LIN {X 0,Y 190.994,Z 614.523,A -85,B 0,C 180,E1 -21873.163,E2 -21873.163} C_VEL
LIN {X 0,Y 190.359,Z 618.573,A -85,B 0,C 180,E1 -21876.358,E2 -21876.358} C_VEL
LIN {X 0,Y 189.98,Z 620.669,A -85,B 0,C 180,E1 -21878.509,E2 -21878.509} C_VEL
LIN {X 0,Y 189.805,Z 622.334,A -85,B 0,C 180,E1 -21880.668,E2 -21880.668} C_VEL
LIN {X 0,Y 189.783,Z 623.59,A -85,B 0,C 180,E1 -21882.837,E2 -21882.837} C_VEL
LIN {X 0,Y 189.941,Z 624.591,A -85,B 0,C 180,E1 -21885.84,E2 -21885.84} C_VEL
LIN {X 0,Y 190.376,Z 624.78,A -85,B 0,C 180,E1 -21889.404,E2 -21889.404} C_VEL
LIN {X 0,Y 191.476,Z 623.671,A -85,B 0,C 180,E1 -21893.421,E2 -21893.421} C_VEL
LIN {X 0,Y 192.56,Z 622.169,A -85,B 0,C 180,E1 -21895.973,E2 -21895.973} C_VEL
LIN {X 0,Y 194.335,Z 619.447,A -85,B 0,C 180,E1 -21899.131,E2 -21899.131} C_VEL
LIN {X 0,Y 196.821,Z 615.459,A -85,B 0,C 180,E1 -21902.384,E2 -21902.384} C_VEL
LIN {X 0,Y 199.68,Z 610.497,A -85,B 0,C 180,E1 -21905.398,E2 -21905.398} C_VEL
LIN {X 0,Y 203.214,Z 603.837,A -85,B 0,C 180,E1 -21908.499,E2 -21908.499} C_VEL
LIN {X 0,Y 207.18,Z 595.882,A -85,B 0,C 180,E1 -21911.297,E2 -21911.297} C_VEL
LIN {X 0,Y 211.109,Z 587.168,A -85,B 0,C 180,E1 -21913.691,E2 -21913.691} C_VEL
LIN {X 0,Y 215.19,Z 576.766,A -85,B 0,C 180,E1 -21915.93,E2 -21915.93} C_VEL
LIN {X 0,Y 218.717,Z 566.352,A -85,B 0,C 180,E1 -21917.649,E2 -21917.649} C_VEL
LIN {X 0,Y 221.86,Z 554.889,A -85,B 0,C 180,E1 -21919.137,E2 -21919.137} C_VEL
LIN {X 0,Y 224.521,Z 543.286,A -85,B 0,C 180,E1 -21920.249,E2 -21920.249} C_VEL
LIN {X 0,Y 226.733,Z 530.168,A -85,B 0,C 180,E1 -21921.135,E2 -21921.135} C_VEL
LIN {X 0,Y 228.18,Z 516.758,A -85,B 0,C 180,E1 -21921.695,E2 -21921.695} C_VEL
LIN {X 0,Y 230.429,Z 476.831,A -85,B 0,C 180,E1 -21922.898,E2 -21922.898} C_VEL
LIN {X 0,Y 225.493,Z 465.84,A -85,B 0,C 180,E1 -21924.695,E2 -21924.695} C_VEL
LIN {X 0,Y 218.885,Z 453.171,A -85,B 0,C 180,E1 -21927.233,E2 -21927.233} C_VEL
LIN {X 0,Y 213.425,Z 444.071,A -85,B 0,C 180,E1 -21929.489,E2 -21929.489} C_VEL
LIN {X 0,Y 207.886,Z 435.651,A -85,B 0,C 180,E1 -21931.986,E2 -21931.986} C_VEL
LIN {X 0,Y 204.807,Z 431.149,A -85,B 0,C 180,E1 -21933.507,E2 -21933.507} C_VEL
LIN {X 0,Y 201.32,Z 426.295,A -85,B 0,C 180,E1 -21935.361,E2 -21935.361} C_VEL
LIN {X 0,Y 198.268,Z 423.081,A -85,B 0,C 180,E1 -21937.051,E2 -21937.051} C_VEL
LIN {X 0,Y 197.017,Z 420.675,A -85,B 0,C 180,E1 -21937.865,E2 -21937.865} C_VEL
LIN {X 0,Y 194.483,Z 418.918,A -85,B 0,C 180,E1 -21939.37,E2 -21939.37} C_VEL
LIN {X 0,Y 193.045,Z 416.552,A -85,B 0,C 180,E1 -21940.39,E2 -21940.39} C_VEL
LIN {X 0,Y 192.687,Z 414.988,A -85,B 0,C 180,E1 -21940.947,E2 -21940.947} C_VEL
LIN {X 0,Y 192.766,Z 414.961,A -85,B 0,C 180,E1 -21945.214,E2 -21945.214} C_VEL
LIN {X 0,Y 192.977,Z 414.933,A -85,B 0,C 180,E1 -21949.508,E2 -21949.508} C_VEL
LIN {X 0,Y 193.063,Z 414.934,A -85,B 0,C 180,E1 -21951.628,E2 -21951.628} C_VEL
LIN {X 0,Y 193.285,Z 414.897,A -85,B 0,C 180,E1 -21957.916,E2 -21957.916} C_VEL
LIN {X 0,Y 193.441,Z 414.876,A -85,B 0,C 180,E1 -21960,E2 -21960} C_VEL
LIN {X 0,Y 192.974,Z 414.931,A -85,B 0,C 180,E1 -21964.177,E2 -21964.177} C_VEL
LIN {X 0,Y 193.057,Z 414.921,A -85,B 0,C 180,E1 -21968.373,E2 -21968.373} C_VEL
LIN {X 0,Y 192.848,Z 414.95,A -85,B 0,C 180,E1 -21972.631,E2 -21972.631} C_VEL
LIN {X 0,Y 192.754,Z 414.966,A -85,B 0,C 180,E1 -21976.959,E2 -21976.959} C_VEL
LIN {X 0,Y 192.632,Z 414.982,A -85,B 0,C 180,E1 -21981.398,E2 -21981.398} C_VEL
LIN {X 0,Y 192.66,Z 414.98,A -85,B 0,C 180,E1 -21984.225,E2 -21984.225} C_VEL
LIN {X 0,Y 192.637,Z 414.994,A -85,B 0,C 180,E1 -21989.825,E2 -21989.825} C_VEL
LIN {X 0,Y 193.264,Z 417.133,A -85,B 0,C 180,E1 -21992.447,E2 -21992.447} C_VEL
LIN {X 0,Y 196.392,Z 421.792,A -85,B 0,C 180,E1 -21994.742,E2 -21994.742} C_VEL
LIN {X 0,Y 198.523,Z 424.312,A -85,B 0,C 180,E1 -21996.017,E2 -21996.017} C_VEL
LIN {X 0,Y 201.888,Z 428.904,A -85,B 0,C 180,E1 -21997.926,E2 -21997.926} C_VEL
LIN {X 0,Y 206.788,Z 436.093,A -85,B 0,C 180,E1 -22000.461,E2 -22000.461} C_VEL
LIN {X 0,Y 210.846,Z 442.58,A -85,B 0,C 180,E1 -22002.372,E2 -22002.372} C_VEL
LIN {X 0,Y 213.909,Z 447.532,A -85,B 0,C 180,E1 -22003.715,E2 -22003.715} C_VEL
LIN {X 0,Y 218.741,Z 455.989,A -85,B 0,C 180,E1 -22005.716,E2 -22005.716} C_VEL
LIN {X 0,Y 223.354,Z 464.921,A -85,B 0,C 180,E1 -22007.517,E2 -22007.517} C_VEL
LIN {X 0,Y 228.843,Z 477.071,A -85,B 0,C 180,E1 -22009.561,E2 -22009.561} C_VEL
LIN {X 0,Y 230.311,Z 480.688,A -85,B 0,C 180,E1 -22010.095,E2 -22010.095} C_VEL
LIN {X 0,Y 229.964,Z 487.939,A -85,B 0,C 180,E1 -22010.327,E2 -22010.327} C_VEL
LIN {X 0,Y 229.156,Z 493.792,A -85,B 0,C 180,E1 -22010.382,E2 -22010.382} C_VEL
LIN {X 0,Y 223.837,Z 512.829,A -85,B 0,C 180,E1 -22009.876,E2 -22009.876} C_VEL
LIN {X 0,Y 223.075,Z 518.674,A -85,B 0,C 180,E1 -22009.947,E2 -22009.947} C_VEL
LIN {X 0,Y 221.839,Z 531.752,A -85,B 0,C 180,E1 -22010.449,E2 -22010.449} C_VEL
LIN {X 0,Y 219.711,Z 544.896,A -85,B 0,C 180,E1 -22011.264,E2 -22011.264} C_VEL
LIN {X 0,Y 216.997,Z 556.869,A -85,B 0,C 180,E1 -22012.317,E2 -22012.317} C_VEL
LIN {X 0,Y 214.084,Z 566.962,A -85,B 0,C 180,E1 -22013.488,E2 -22013.488} C_VEL
LIN {X 0,Y 210.527,Z 577.729,A -85,B 0,C 180,E1 -22015.134,E2 -22015.134} C_VEL
LIN {X 0,Y 206.719,Z 587.501,A -85,B 0,C 180,E1 -22017.047,E2 -22017.047} C_VEL
LIN {X 0,Y 202.701,Z 596.411,A -85,B 0,C 180,E1 -22019.244,E2 -22019.244} C_VEL
LIN {X 0,Y 198.334,Z 605.127,A -85,B 0,C 180,E1 -22021.998,E2 -22021.998} C_VEL
LIN {X 0,Y 194.658,Z 612.111,A -85,B 0,C 180,E1 -22024.899,E2 -22024.899} C_VEL
LIN {X 0,Y 190.924,Z 618.518,A -85,B 0,C 180,E1 -22028.402,E2 -22028.402} C_VEL
LIN {X 0,Y 188.197,Z 622.767,A -85,B 0,C 180,E1 -22031.494,E2 -22031.494} C_VEL
LIN {X 0,Y 186.158,Z 625.973,A -85,B 0,C 180,E1 -22034.677,E2 -22034.677} C_VEL
LIN {X 0,Y 184.265,Z 628.793,A -85,B 0,C 180,E1 -22039.007,E2 -22039.007} C_VEL
LIN {X 0,Y 183.303,Z 629.978,A -85,B 0,C 180,E1 -22043.396,E2 -22043.396} C_VEL
LIN {X 0,Y 183.013,Z 629.839,A -85,B 0,C 180,E1 -22046.809,E2 -22046.809} C_VEL
LIN {X 0,Y 183.082,Z 628.864,A -85,B 0,C 180,E1 -22050.001,E2 -22050.001} C_VEL
LIN {X 0,Y 183.013,Z 627.001,A -85,B 0,C 180,E1 -22053.192,E2 -22053.192} C_VEL
LIN {X 0,Y 183.21,Z 624.002,A -85,B 0,C 180,E1 -22056.609,E2 -22056.609} C_VEL
LIN {X 0,Y 183.741,Z 620.023,A -85,B 0,C 180,E1 -22059.912,E2 -22059.912} C_VEL
LIN {X 0,Y 184.859,Z 613.872,A -85,B 0,C 180,E1 -22063.746,E2 -22063.746} C_VEL
LIN {X 0,Y 186.434,Z 607.134,A -85,B 0,C 180,E1 -22066.987,E2 -22066.987} C_VEL
LIN {X 0,Y 188.49,Z 598.75,A -85,B 0,C 180,E1 -22070.175,E2 -22070.175} C_VEL
LIN {X 0,Y 190.515,Z 589.828,A -85,B 0,C 180,E1 -22072.863,E2 -22072.863} C_VEL
LIN {X 0,Y 192.86,Z 579.376,A -85,B 0,C 180,E1 -22075.352,E2 -22075.352} C_VEL
LIN {X 0,Y 195.074,Z 568.74,A -85,B 0,C 180,E1 -22077.345,E2 -22077.345} C_VEL
LIN {X 0,Y 197.308,Z 556.933,A -85,B 0,C 180,E1 -22079.033,E2 -22079.033} C_VEL
LIN {X 0,Y 199.073,Z 544.595,A -85,B 0,C 180,E1 -22080.35,E2 -22080.35} C_VEL
LIN {X 0,Y 200.455,Z 532.006,A -85,B 0,C 180,E1 -22081.287,E2 -22081.287} C_VEL
LIN {X 0,Y 201.278,Z 519.169,A -85,B 0,C 180,E1 -22081.876,E2 -22081.876} C_VEL
LIN {X 0,Y 203.223,Z 469.686,A -85,B 0,C 180,E1 -22083.552,E2 -22083.552} C_VEL
LIN {X 0,Y 201.364,Z 454.761,A -85,B 0,C 180,E1 -22084.437,E2 -22084.437} C_VEL
LIN {X 0,Y 195.911,Z 439.957,A -85,B 0,C 180,E1 -22085.949,E2 -22085.949} C_VEL
LIN {X 0,Y 189.605,Z 425.442,A -85,B 0,C 180,E1 -22087.713,E2 -22087.713} C_VEL
LIN {X 0,Y 186.159,Z 418.355,A -85,B 0,C 180,E1 -22088.776,E2 -22088.776} C_VEL
LIN {X 0,Y 185.522,Z 415.966,A -85,B 0,C 180,E1 -22090.09,E2 -22090.09} C_VEL
LIN {X 0,Y 185.538,Z 415.833,A -85,B 0,C 180,E1 -22093.97,E2 -22093.97} C_VEL
LIN {X 0,Y 185.557,Z 415.82,A -85,B 0,C 180,E1 -22097.019,E2 -22097.019} C_VEL
LIN {X 0,Y 185.542,Z 415.866,A -85,B 0,C 180,E1 -22099.914,E2 -22099.914} C_VEL
LIN {X 0,Y 185.56,Z 415.861,A -85,B 0,C 180,E1 -22102.699,E2 -22102.699} C_VEL
LIN {X 0,Y 185.541,Z 415.875,A -85,B 0,C 180,E1 -22107.974,E2 -22107.974} C_VEL
LIN {X 0,Y 185.58,Z 415.848,A -85,B 0,C 180,E1 -22110.576,E2 -22110.576} C_VEL
LIN {X 0,Y 185.579,Z 415.87,A -85,B 0,C 180,E1 -22115.381,E2 -22115.381} C_VEL
LIN {X 0,Y 185.672,Z 415.834,A -85,B 0,C 180,E1 -22121.135,E2 -22121.135} C_VEL
LIN {X 0,Y 185.693,Z 415.854,A -85,B 0,C 180,E1 -22124.637,E2 -22124.637} C_VEL
LIN {X 0,Y 185.887,Z 415.794,A -85,B 0,C 180,E1 -22129.418,E2 -22129.418} C_VEL
LIN {X 0,Y 185.946,Z 415.817,A -85,B 0,C 180,E1 -22133.489,E2 -22133.489} C_VEL
LIN {X 0,Y 186.205,Z 415.778,A -85,B 0,C 180,E1 -22137.837,E2 -22137.837} C_VEL
LIN {X 0,Y 186.405,Z 415.728,A -85,B 0,C 180,E1 -22140,E2 -22140} C_VEL
LIN {X 0,Y 185.919,Z 415.816,A -85,B 0,C 180,E1 -22144.336,E2 -22144.336} C_VEL
LIN {X 0,Y 185.985,Z 415.81,A -85,B 0,C 180,E1 -22148.694,E2 -22148.694} C_VEL
LIN {X 0,Y 185.727,Z 415.81,A -85,B 0,C 180,E1 -22153.123,E2 -22153.123} C_VEL
LIN {X 0,Y 185.688,Z 415.855,A -85,B 0,C 180,E1 -22157.625,E2 -22157.625} C_VEL
LIN {X 0,Y 185.595,Z 415.836,A -85,B 0,C 180,E1 -22162.251,E2 -22162.251} C_VEL
LIN {X 0,Y 185.561,Z 415.861,A -85,B 0,C 180,E1 -22167.032,E2 -22167.032} C_VEL
LIN {X 0,Y 185.578,Z 415.866,A -85,B 0,C 180,E1 -22169.493,E2 -22169.493} C_VEL
LIN {X 0,Y 185.499,Z 415.851,A -85,B 0,C 180,E1 -22174.632,E2 -22174.632} C_VEL
LIN {X 0,Y 185.505,Z 415.876,A -85,B 0,C 180,E1 -22177.313,E2 -22177.313} C_VEL
LIN {X 0,Y 185.471,Z 415.863,A -85,B 0,C 180,E1 -22180.725,E2 -22180.725} C_VEL
LIN {X 0,Y 185.514,Z 415.877,A -85,B 0,C 180,E1 -22186.037,E2 -22186.037} C_VEL
LIN {X 0,Y 185.535,Z 415.86,A -85,B 0,C 180,E1 -22189.913,E2 -22189.913} C_VEL
LIN {X 0,Y 185.56,Z 415.873,A -85,B 0,C 180,E1 -22192.7,E2 -22192.7} C_VEL
LIN {X 0,Y 185.545,Z 415.82,A -85,B 0,C 180,E1 -22197.975,E2 -22197.975} C_VEL
LIN {X 0,Y 185.583,Z 415.851,A -85,B 0,C 180,E1 -22200.576,E2 -22200.576} C_VEL
LIN {X 0,Y 185.588,Z 416.049,A -85,B 0,C 180,E1 -22203.984,E2 -22203.984} C_VEL
LIN {X 0,Y 185.857,Z 417.152,A -85,B 0,C 180,E1 -22204.408,E2 -22204.408} C_VEL
LIN {X 0,Y 192.547,Z 429.043,A -85,B 0,C 180,E1 -22206.245,E2 -22206.245} C_VEL
LIN {X 0,Y 199.331,Z 445.451,A -85,B 0,C 180,E1 -22208.111,E2 -22208.111} C_VEL
LIN {X 0,Y 203.23,Z 457.05,A -85,B 0,C 180,E1 -22209.202,E2 -22209.202} C_VEL
LIN {X 0,Y 203.683,Z 460.656,A -85,B 0,C 180,E1 -22209.415,E2 -22209.415} C_VEL
LIN {X 0,Y 200.97,Z 521.074,A -85,B 0,C 180,E1 -22211.465,E2 -22211.465} C_VEL
LIN {X 0,Y 199.777,Z 534.184,A -85,B 0,C 180,E1 -22212.271,E2 -22212.271} C_VEL
LIN {X 0,Y 198.333,Z 545.664,A -85,B 0,C 180,E1 -22213.32,E2 -22213.32} C_VEL
LIN {X 0,Y 196.576,Z 557.28,A -85,B 0,C 180,E1 -22214.769,E2 -22214.769} C_VEL
LIN {X 0,Y 194.246,Z 568.912,A -85,B 0,C 180,E1 -22216.664,E2 -22216.664} C_VEL
LIN {X 0,Y 192.061,Z 578.513,A -85,B 0,C 180,E1 -22218.657,E2 -22218.657} C_VEL
LIN {X 0,Y 190.061,Z 587.384,A -85,B 0,C 180,E1 -22220.958,E2 -22220.958} C_VEL
LIN {X 0,Y 188.135,Z 595.539,A -85,B 0,C 180,E1 -22223.565,E2 -22223.565} C_VEL
LIN {X 0,Y 186.174,Z 603.553,A -85,B 0,C 180,E1 -22226.753,E2 -22226.753} C_VEL
LIN {X 0,Y 184.788,Z 609.949,A -85,B 0,C 180,E1 -22229.999,E2 -22229.999} C_VEL
LIN {X 0,Y 183.854,Z 615.031,A -85,B 0,C 180,E1 -22233.286,E2 -22233.286} C_VEL
LIN {X 0,Y 183.202,Z 618.982,A -85,B 0,C 180,E1 -22236.608,E2 -22236.608} C_VEL
LIN {X 0,Y 182.852,Z 621.023,A -85,B 0,C 180,E1 -22238.843,E2 -22238.843} C_VEL
LIN {X 0,Y 182.68,Z 622.642,A -85,B 0,C 180,E1 -22241.09,E2 -22241.09} C_VEL
LIN {X 0,Y 182.711,Z 623.832,A -85,B 0,C 180,E1 -22243.343,E2 -22243.343} C_VEL
LIN {X 0,Y 182.855,Z 624.677,A -85,B 0,C 180,E1 -22246.082,E2 -22246.082} C_VEL
LIN {X 0,Y 183.415,Z 624.861,A -85,B 0,C 180,E1 -22250.172,E2 -22250.172} C_VEL
LIN {X 0,Y 184.509,Z 623.825,A -85,B 0,C 180,E1 -22253.913,E2 -22253.913} C_VEL
LIN {X 0,Y 185.902,Z 622.066,A -85,B 0,C 180,E1 -22256.977,E2 -22256.977} C_VEL
LIN {X 0,Y 188.322,Z 618.585,A -85,B 0,C 180,E1 -22260.87,E2 -22260.87} C_VEL
LIN {X 0,Y 191.556,Z 613.535,A -85,B 0,C 180,E1 -22264.657,E2 -22264.657} C_VEL
LIN {X 0,Y 194.896,Z 607.847,A -85,B 0,C 180,E1 -22267.807,E2 -22267.807} C_VEL
LIN {X 0,Y 198.852,Z 600.683,A -85,B 0,C 180,E1 -22270.83,E2 -22270.83} C_VEL
LIN {X 0,Y 202.502,Z 593.434,A -85,B 0,C 180,E1 -22273.212,E2 -22273.212} C_VEL
LIN {X 0,Y 207.074,Z 583.27,A -85,B 0,C 180,E1 -22275.803,E2 -22275.803} C_VEL
LIN {X 0,Y 210.804,Z 573.718,A -85,B 0,C 180,E1 -22277.703,E2 -22277.703} C_VEL
LIN {X 0,Y 214.284,Z 563.353,A -85,B 0,C 180,E1 -22279.325,E2 -22279.325} C_VEL
LIN {X 0,Y 217.324,Z 551.943,A -85,B 0,C 180,E1 -22280.722,E2 -22280.722} C_VEL
LIN {X 0,Y 220.163,Z 539.25,A -85,B 0,C 180,E1 -22281.818,E2 -22281.818} C_VEL
LIN {X 0,Y 222.158,Z 526.661,A -85,B 0,C 180,E1 -22282.578,E2 -22282.578} C_VEL
LIN {X 0,Y 223.409,Z 512.666,A -85,B 0,C 180,E1 -22283.092,E2 -22283.092} C_VEL
LIN {X 0,Y 225.409,Z 479.362,A -85,B 0,C 180,E1 -22284.09,E2 -22284.09} C_VEL
LIN {X 0,Y 219.955,Z 467.378,A -85,B 0,C 180,E1 -22286.201,E2 -22286.201} C_VEL
LIN {X 0,Y 213.949,Z 455.886,A -85,B 0,C 180,E1 -22288.675,E2 -22288.675} C_VEL
LIN {X 0,Y 208.169,Z 446.321,A -85,B 0,C 180,E1 -22291.252,E2 -22291.252} C_VEL
LIN {X 0,Y 202.246,Z 437.272,A -85,B 0,C 180,E1 -22294.216,E2 -22294.216} C_VEL
LIN {X 0,Y 198.374,Z 431.996,A -85,B 0,C 180,E1 -22296.363,E2 -22296.363} C_VEL
LIN {X 0,Y 195.724,Z 428.998,A -85,B 0,C 180,E1 -22297.92,E2 -22297.92} C_VEL
LIN {X 0,Y 194.566,Z 427.074,A -85,B 0,C 180,E1 -22298.687,E2 -22298.687} C_VEL
LIN {X 0,Y 191.883,Z 424.685,A -85,B 0,C 180,E1 -22300.406,E2 -22300.406} C_VEL
LIN {X 0,Y 190.206,Z 421.606,A -85,B 0,C 180,E1 -22301.7,E2 -22301.7} C_VEL
LIN {X 0,Y 187.509,Z 419.777,A -85,B 0,C 180,E1 -22303.674,E2 -22303.674} C_VEL
LIN {X 0,Y 186.147,Z 417.583,A -85,B 0,C 180,E1 -22304.886,E2 -22304.886} C_VEL
LIN {X 0,Y 185.716,Z 415.838,A -85,B 0,C 180,E1 -22305.481,E2 -22305.481} C_VEL
LIN {X 0,Y 185.92,Z 415.812,A -85,B 0,C 180,E1 -22309.359,E2 -22309.359} C_VEL
LIN {X 0,Y 185.962,Z 415.808,A -85,B 0,C 180,E1 -22313.49,E2 -22313.49} C_VEL
LIN {X 0,Y 186.226,Z 415.777,A -85,B 0,C 180,E1 -22317.837,E2 -22317.837} C_VEL
LIN {X 0,Y 186.405,Z 415.752,A -85,B 0,C 180,E1 -22320,E2 -22320} C_VEL
LIN {X 0,Y 185.921,Z 415.809,A -85,B 0,C 180,E1 -22324.336,E2 -22324.336} C_VEL
LIN {X 0,Y 186.004,Z 415.799,A -85,B 0,C 180,E1 -22328.693,E2 -22328.693} C_VEL
LIN {X 0,Y 185.759,Z 415.83,A -85,B 0,C 180,E1 -22333.121,E2 -22333.121} C_VEL
LIN {X 0,Y 185.686,Z 415.841,A -85,B 0,C 180,E1 -22337.626,E2 -22337.626} C_VEL
LIN {X 0,Y 185.592,Z 415.853,A -85,B 0,C 180,E1 -22342.252,E2 -22342.252} C_VEL
LIN {X 0,Y 185.595,Z 416.077,A -85,B 0,C 180,E1 -22346.343,E2 -22346.343} C_VEL
LIN {X 0,Y 185.883,Z 417.248,A -85,B 0,C 180,E1 -22347.591,E2 -22347.591} C_VEL
LIN {X 0,Y 187.793,Z 420.157,A -85,B 0,C 180,E1 -22349.412,E2 -22349.412} C_VEL
LIN {X 0,Y 191.541,Z 424.344,A -85,B 0,C 180,E1 -22352.213,E2 -22352.213} C_VEL
LIN {X 0,Y 194.377,Z 428.316,A -85,B 0,C 180,E1 -22354.158,E2 -22354.158} C_VEL
LIN {X 0,Y 196.063,Z 430.428,A -85,B 0,C 180,E1 -22355.215,E2 -22355.215} C_VEL
LIN {X 0,Y 200.345,Z 436.508,A -85,B 0,C 180,E1 -22357.733,E2 -22357.733} C_VEL
LIN {X 0,Y 204.101,Z 442.27,A -85,B 0,C 180,E1 -22359.748,E2 -22359.748} C_VEL
LIN {X 0,Y 209.575,Z 451.128,A -85,B 0,C 180,E1 -22362.396,E2 -22362.396} C_VEL
LIN {X 0,Y 215.024,Z 460.924,A -85,B 0,C 180,E1 -22364.795,E2 -22364.795} C_VEL
LIN {X 0,Y 219.601,Z 470.072,A -85,B 0,C 180,E1 -22366.679,E2 -22366.679} C_VEL
LIN {X 0,Y 224.654,Z 481.579,A -85,B 0,C 180,E1 -22368.661,E2 -22368.661} C_VEL
LIN {X 0,Y 225.232,Z 483.09,A -85,B 0,C 180,E1 -22368.886,E2 -22368.886} C_VEL
LIN {X 0,Y 223.075,Z 518.674,A -85,B 0,C 180,E1 -22369.947,E2 -22369.947} C_VEL
LIN {X 0,Y 222.23,Z 524.511,A -85,B 0,C 180,E1 -22370.032,E2 -22370.032} C_VEL
LIN {X 0,Y 219.097,Z 533.93,A -85,B 0,C 180,E1 -22369.922,E2 -22369.922} C_VEL
LIN {X 0,Y 215.487,Z 543.165,A -85,B 0,C 180,E1 -22369.943,E2 -22369.943} C_VEL
LIN {X 0,Y 213.894,Z 548.708,A -85,B 0,C 180,E1 -22370.266,E2 -22370.266} C_VEL
LIN {X 0,Y 210.421,Z 561.705,A -85,B 0,C 180,E1 -22371.534,E2 -22371.534} C_VEL
LIN {X 0,Y 207.042,Z 572.248,A -85,B 0,C 180,E1 -22372.951,E2 -22372.951} C_VEL
LIN {X 0,Y 203.003,Z 583.035,A -85,B 0,C 180,E1 -22374.862,E2 -22374.862} C_VEL
LIN {X 0,Y 198.297,Z 593.626,A -85,B 0,C 180,E1 -22377.285,E2 -22377.285} C_VEL
LIN {X 0,Y 194.287,Z 601.461,A -85,B 0,C 180,E1 -22379.575,E2 -22379.575} C_VEL
LIN {X 0,Y 190.24,Z 608.929,A -85,B 0,C 180,E1 -22382.389,E2 -22382.389} C_VEL
LIN {X 0,Y 186.497,Z 615.305,A -85,B 0,C 180,E1 -22385.512,E2 -22385.512} C_VEL
LIN {X 0,Y 183.306,Z 620.235,A -85,B 0,C 180,E1 -22388.641,E2 -22388.641} C_VEL
LIN {X 0,Y 180.632,Z 624.061,A -85,B 0,C 180,E1 -22391.866,E2 -22391.866} C_VEL
LIN {X 0,Y 178.159,Z 627.614,A -85,B 0,C 180,E1 -22396.31,E2 -22396.31} C_VEL
LIN {X 0,Y 177.282,Z 628.785,A -85,B 0,C 180,E1 -22398.568,E2 -22398.568} C_VEL
LIN {X 0,Y 176.243,Z 629.892,A -85,B 0,C 180,E1 -22403.13,E2 -22403.13} C_VEL
LIN {X 0,Y 175.912,Z 629.589,A -85,B 0,C 180,E1 -22407.196,E2 -22407.196} C_VEL
LIN {X 0,Y 175.993,Z 628.659,A -85,B 0,C 180,E1 -22410.001,E2 -22410.001} C_VEL
LIN {X 0,Y 175.912,Z 627.093,A -85,B 0,C 180,E1 -22412.805,E2 -22412.805} C_VEL
LIN {X 0,Y 176.137,Z 623.691,A -85,B 0,C 180,E1 -22416.875,E2 -22416.875} C_VEL
LIN {X 0,Y 176.71,Z 619.644,A -85,B 0,C 180,E1 -22420.31,E2 -22420.31} C_VEL
LIN {X 0,Y 177.931,Z 613.392,A -85,B 0,C 180,E1 -22424.292,E2 -22424.292} C_VEL
LIN {X 0,Y 179.6,Z 606.568,A -85,B 0,C 180,E1 -22427.654,E2 -22427.654} C_VEL
LIN {X 0,Y 181.827,Z 598.061,A -85,B 0,C 180,E1 -22430.949,E2 -22430.949} C_VEL
LIN {X 0,Y 184.036,Z 588.508,A -85,B 0,C 180,E1 -22433.862,E2 -22433.862} C_VEL
LIN {X 0,Y 186.395,Z 578.387,A -85,B 0,C 180,E1 -22436.298,E2 -22436.298} C_VEL
LIN {X 0,Y 188.782,Z 567.541,A -85,B 0,C 180,E1 -22438.337,E2 -22438.337} C_VEL
LIN {X 0,Y 191.074,Z 555.334,A -85,B 0,C 180,E1 -22440.076,E2 -22440.076} C_VEL
LIN {X 0,Y 192.925,Z 542.538,A -85,B 0,C 180,E1 -22441.425,E2 -22441.425} C_VEL
LIN {X 0,Y 194.304,Z 529.879,A -85,B 0,C 180,E1 -22442.319,E2 -22442.319} C_VEL
LIN {X 0,Y 195.232,Z 512.784,A -85,B 0,C 180,E1 -22443.026,E2 -22443.026} C_VEL
LIN {X 0,Y 196.968,Z 470.347,A -85,B 0,C 180,E1 -22444.503,E2 -22444.503} C_VEL
LIN {X 0,Y 195.349,Z 457.02,A -85,B 0,C 180,E1 -22445.326,E2 -22445.326} C_VEL
LIN {X 0,Y 189.914,Z 442.19,A -85,B 0,C 180,E1 -22446.924,E2 -22446.924} C_VEL
LIN {X 0,Y 183.723,Z 428.101,A -85,B 0,C 180,E1 -22448.756,E2 -22448.756} C_VEL
LIN {X 0,Y 178.82,Z 418.225,A -85,B 0,C 180,E1 -22450.346,E2 -22450.346} C_VEL
LIN {X 0,Y 178.475,Z 416.838,A -85,B 0,C 180,E1 -22451.139,E2 -22451.139} C_VEL
LIN {X 0,Y 178.49,Z 416.697,A -85,B 0,C 180,E1 -22455.133,E2 -22455.133} C_VEL
LIN {X 0,Y 178.502,Z 416.713,A -85,B 0,C 180,E1 -22458.423,E2 -22458.423} C_VEL
LIN {X 0,Y 178.459,Z 416.738,A -85,B 0,C 180,E1 -22463.791,E2 -22463.791} C_VEL
LIN {X 0,Y 178.49,Z 416.752,A -85,B 0,C 180,E1 -22466.547,E2 -22466.547} C_VEL
LIN {X 0,Y 178.521,Z 416.73,A -85,B 0,C 180,E1 -22470.007,E2 -22470.007} C_VEL
LIN {X 0,Y 178.519,Z 416.748,A -85,B 0,C 180,E1 -22474.886,E2 -22474.886} C_VEL
LIN {X 0,Y 178.62,Z 416.708,A -85,B 0,C 180,E1 -22480.786,E2 -22480.786} C_VEL
LIN {X 0,Y 178.656,Z 416.723,A -85,B 0,C 180,E1 -22486.347,E2 -22486.347} C_VEL
LIN {X 0,Y 178.91,Z 416.667,A -85,B 0,C 180,E1 -22490.959,E2 -22490.959} C_VEL
LIN {X 0,Y 178.866,Z 416.705,A -85,B 0,C 180,E1 -22495.493,E2 -22495.493} C_VEL
LIN {X 0,Y 179.368,Z 416.603,A -85,B 0,C 180,E1 -22500,E2 -22500} C_VEL
LIN {X 0,Y 178.867,Z 416.696,A -85,B 0,C 180,E1 -22504.507,E2 -22504.507} C_VEL
LIN {X 0,Y 178.913,Z 416.687,A -85,B 0,C 180,E1 -22509.04,E2 -22509.04} C_VEL
LIN {X 0,Y 178.655,Z 416.692,A -85,B 0,C 180,E1 -22513.652,E2 -22513.652} C_VEL
LIN {X 0,Y 178.622,Z 416.732,A -85,B 0,C 180,E1 -22519.216,E2 -22519.216} C_VEL
LIN {X 0,Y 178.524,Z 416.715,A -85,B 0,C 180,E1 -22525.117,E2 -22525.117} C_VEL
LIN {X 0,Y 178.5,Z 416.739,A -85,B 0,C 180,E1 -22530.786,E2 -22530.786} C_VEL
LIN {X 0,Y 178.484,Z 416.721,A -85,B 0,C 180,E1 -22534.219,E2 -22534.219} C_VEL
LIN {X 0,Y 178.395,Z 416.76,A -85,B 0,C 180,E1 -22539.074,E2 -22539.074} C_VEL
LIN {X 0,Y 178.408,Z 416.736,A -85,B 0,C 180,E1 -22542.042,E2 -22542.042} C_VEL
LIN {X 0,Y 178.429,Z 416.758,A -85,B 0,C 180,E1 -22545.152,E2 -22545.152} C_VEL
LIN {X 0,Y 178.448,Z 416.741,A -85,B 0,C 180,E1 -22548.443,E2 -22548.443} C_VEL
LIN {X 0,Y 178.489,Z 416.755,A -85,B 0,C 180,E1 -22551.952,E2 -22551.952} C_VEL
LIN {X 0,Y 178.491,Z 416.697,A -85,B 0,C 180,E1 -22556.548,E2 -22556.548} C_VEL
LIN {X 0,Y 178.514,Z 416.747,A -85,B 0,C 180,E1 -22561.808,E2 -22561.808} C_VEL
LIN {X 0,Y 178.555,Z 417.072,A -85,B 0,C 180,E1 -22562.617,E2 -22562.617} C_VEL
LIN {X 0,Y 178.966,Z 418.482,A -85,B 0,C 180,E1 -22563.019,E2 -22563.019} C_VEL
LIN {X 0,Y 184.777,Z 428.314,A -85,B 0,C 180,E1 -22564.722,E2 -22564.722} C_VEL
LIN {X 0,Y 188.631,Z 436.049,A -85,B 0,C 180,E1 -22565.821,E2 -22565.821} C_VEL
LIN {X 0,Y 194.868,Z 451.953,A -85,B 0,C 180,E1 -22567.634,E2 -22567.634} C_VEL
LIN {X 0,Y 197.222,Z 459.48,A -85,B 0,C 180,E1 -22568.344,E2 -22568.344} C_VEL
LIN {X 0,Y 197.306,Z 464.411,A -85,B 0,C 180,E1 -22568.562,E2 -22568.562} C_VEL
LIN {X 0,Y 194.668,Z 520.834,A -85,B 0,C 180,E1 -22570.523,E2 -22570.523} C_VEL
LIN {X 0,Y 193.434,Z 534.023,A -85,B 0,C 180,E1 -22571.347,E2 -22571.347} C_VEL
LIN {X 0,Y 191.899,Z 545.725,A -85,B 0,C 180,E1 -22572.439,E2 -22572.439} C_VEL
LIN {X 0,Y 189.955,Z 557.989,A -85,B 0,C 180,E1 -22574.021,E2 -22574.021} C_VEL
LIN {X 0,Y 187.626,Z 569.126,A -85,B 0,C 180,E1 -22575.908,E2 -22575.908} C_VEL
LIN {X 0,Y 185.355,Z 578.708,A -85,B 0,C 180,E1 -22577.963,E2 -22577.963} C_VEL
LIN {X 0,Y 183.011,Z 588.463,A -85,B 0,C 180,E1 -22580.606,E2 -22580.606} C_VEL
LIN {X 0,Y 181.083,Z 596.45,A -85,B 0,C 180,E1 -22583.313,E2 -22583.313} C_VEL
LIN {X 0,Y 179.04,Z 604.292,A -85,B 0,C 180,E1 -22586.624,E2 -22586.624} C_VEL
LIN {X 0,Y 177.631,Z 610.548,A -85,B 0,C 180,E1 -22589.999,E2 -22589.999} C_VEL
LIN {X 0,Y 176.721,Z 615.523,A -85,B 0,C 180,E1 -22593.419,E2 -22593.419} C_VEL
LIN {X 0,Y 176.062,Z 619.378,A -85,B 0,C 180,E1 -22596.877,E2 -22596.877} C_VEL
LIN {X 0,Y 175.711,Z 621.373,A -85,B 0,C 180,E1 -22599.206,E2 -22599.206} C_VEL
LIN {X 0,Y 175.564,Z 622.944,A -85,B 0,C 180,E1 -22601.545,E2 -22601.545} C_VEL
LIN {X 0,Y 175.613,Z 624.047,A -85,B 0,C 180,E1 -22603.893,E2 -22603.893} C_VEL
LIN {X 0,Y 175.776,Z 624.763,A -85,B 0,C 180,E1 -22606.345,E2 -22606.345} C_VEL
LIN {X 0,Y 176.039,Z 625.043,A -85,B 0,C 180,E1 -22608.625,E2 -22608.625} C_VEL
LIN {X 0,Y 176.483,Z 624.922,A -85,B 0,C 180,E1 -22611.001,E2 -22611.001} C_VEL
LIN {X 0,Y 177.572,Z 623.97,A -85,B 0,C 180,E1 -22614.453,E2 -22614.453} C_VEL
LIN {X 0,Y 179.293,Z 621.96,A -85,B 0,C 180,E1 -22618.058,E2 -22618.058} C_VEL
LIN {X 0,Y 181.684,Z 618.776,A -85,B 0,C 180,E1 -22621.678,E2 -22621.678} C_VEL
LIN {X 0,Y 184.416,Z 614.841,A -85,B 0,C 180,E1 -22624.863,E2 -22624.863} C_VEL
LIN {X 0,Y 187.999,Z 609.167,A -85,B 0,C 180,E1 -22628.275,E2 -22628.275} C_VEL
LIN {X 0,Y 191.848,Z 602.647,A -85,B 0,C 180,E1 -22631.252,E2 -22631.252} C_VEL
LIN {X 0,Y 195.765,Z 595.439,A -85,B 0,C 180,E1 -22633.82,E2 -22633.82} C_VEL
LIN {X 0,Y 199.811,Z 587.203,A -85,B 0,C 180,E1 -22636.139,E2 -22636.139} C_VEL
LIN {X 0,Y 203.804,Z 577.911,A -85,B 0,C 180,E1 -22638.219,E2 -22638.219} C_VEL
LIN {X 0,Y 207.593,Z 567.88,A -85,B 0,C 180,E1 -22639.966,E2 -22639.966} C_VEL
LIN {X 0,Y 210.994,Z 556.627,A -85,B 0,C 180,E1 -22641.512,E2 -22641.512} C_VEL
LIN {X 0,Y 213.861,Z 545.472,A -85,B 0,C 180,E1 -22642.64,E2 -22642.64} C_VEL
LIN {X 0,Y 216.376,Z 532.408,A -85,B 0,C 180,E1 -22643.599,E2 -22643.599} C_VEL
LIN {X 0,Y 218.03,Z 519.088,A -85,B 0,C 180,E1 -22644.215,E2 -22644.215} C_VEL
LIN {X 0,Y 220.369,Z 481.643,A -85,B 0,C 180,E1 -22645.384,E2 -22645.384} C_VEL
LIN {X 0,Y 215.038,Z 469.947,A -85,B 0,C 180,E1 -22647.582,E2 -22647.582} C_VEL
LIN {X 0,Y 209.42,Z 459.247,A -85,B 0,C 180,E1 -22650.053,E2 -22650.053} C_VEL
LIN {X 0,Y 203.929,Z 450.091,A -85,B 0,C 180,E1 -22652.691,E2 -22652.691} C_VEL
LIN {X 0,Y 199.032,Z 442.516,A -85,B 0,C 180,E1 -22655.318,E2 -22655.318} C_VEL
LIN {X 0,Y 195.787,Z 438.064,A -85,B 0,C 180,E1 -22657.214,E2 -22657.214} C_VEL
LIN {X 0,Y 193.011,Z 434.533,A -85,B 0,C 180,E1 -22658.961,E2 -22658.961} C_VEL
LIN {X 0,Y 192.214,Z 433.405,A -85,B 0,C 180,E1 -22659.5,E2 -22659.5} C_VEL
LIN {X 0,Y 189.463,Z 430.543,A -85,B 0,C 180,E1 -22661.388,E2 -22661.388} C_VEL
LIN {X 0,Y 188.239,Z 428.235,A -85,B 0,C 180,E1 -22662.384,E2 -22662.384} C_VEL
LIN {X 0,Y 185.539,Z 426.067,A -85,B 0,C 180,E1 -22664.483,E2 -22664.483} C_VEL
LIN {X 0,Y 183.977,Z 423.353,A -85,B 0,C 180,E1 -22665.976,E2 -22665.976} C_VEL
LIN {X 0,Y 183.67,Z 422.633,A -85,B 0,C 180,E1 -22666.305,E2 -22666.305} C_VEL
LIN {X 0,Y 180.971,Z 420.956,A -85,B 0,C 180,E1 -22668.934,E2 -22668.934} C_VEL
LIN {X 0,Y 179.422,Z 418.548,A -85,B 0,C 180,E1 -22670.906,E2 -22670.906} C_VEL
LIN {X 0,Y 178.931,Z 416.695,A -85,B 0,C 180,E1 -22671.814,E2 -22671.814} C_VEL
LIN {X 0,Y 179.17,Z 416.656,A -85,B 0,C 180,E1 -22677.752,E2 -22677.752} C_VEL
LIN {X 0,Y 179.368,Z 416.628,A -85,B 0,C 180,E1 -22680,E2 -22680} C_VEL
LIN {X 0,Y 178.869,Z 416.688,A -85,B 0,C 180,E1 -22684.507,E2 -22684.507} C_VEL
LIN {X 0,Y 178.933,Z 416.679,A -85,B 0,C 180,E1 -22689.039,E2 -22689.039} C_VEL
LIN {X 0,Y 178.682,Z 416.711,A -85,B 0,C 180,E1 -22693.65,E2 -22693.65} C_VEL
LIN {X 0,Y 178.646,Z 416.716,A -85,B 0,C 180,E1 -22698.344,E2 -22698.344} C_VEL
LIN {X 0,Y 178.576,Z 416.905,A -85,B 0,C 180,E1 -22700.516,E2 -22700.516} C_VEL
LIN {X 0,Y 179.475,Z 419.468,A -85,B 0,C 180,E1 -22702.142,E2 -22702.142} C_VEL
LIN {X 0,Y 181.446,Z 421.641,A -85,B 0,C 180,E1 -22704.471,E2 -22704.471} C_VEL
LIN {X 0,Y 183.483,Z 423.1,A -85,B 0,C 180,E1 -22706.441,E2 -22706.441} C_VEL
LIN {X 0,Y 186.283,Z 427.004,A -85,B 0,C 180,E1 -22709.003,E2 -22709.003} C_VEL
LIN {X 0,Y 189.406,Z 430.653,A -85,B 0,C 180,E1 -22711.437,E2 -22711.437} C_VEL
LIN {X 0,Y 192.505,Z 434.981,A -85,B 0,C 180,E1 -22713.643,E2 -22713.643} C_VEL
LIN {X 0,Y 194.036,Z 437.181,A -85,B 0,C 180,E1 -22714.656,E2 -22714.656} C_VEL
LIN {X 0,Y 197.626,Z 442.361,A -85,B 0,C 180,E1 -22716.857,E2 -22716.857} C_VEL
LIN {X 0,Y 201.457,Z 448.421,A -85,B 0,C 180,E1 -22719.016,E2 -22719.016} C_VEL
LIN {X 0,Y 206.352,Z 456.63,A -85,B 0,C 180,E1 -22721.512,E2 -22721.512} C_VEL
LIN {X 0,Y 211.867,Z 466.826,A -85,B 0,C 180,E1 -22724.064,E2 -22724.064} C_VEL
LIN {X 0,Y 216.392,Z 476.338,A -85,B 0,C 180,E1 -22726.021,E2 -22726.021} C_VEL
LIN {X 0,Y 220.272,Z 485.439,A -85,B 0,C 180,E1 -22727.624,E2 -22727.624} C_VEL
LIN {X 0,Y 217.45,Z 526.853,A -85,B 0,C 180,E1 -22728.908,E2 -22728.908} C_VEL
LIN {X 0,Y 215.544,Z 540.135,A -85,B 0,C 180,E1 -22729.608,E2 -22729.608} C_VEL
LIN {X 0,Y 213.894,Z 548.708,A -85,B 0,C 180,E1 -22730.266,E2 -22730.266} C_VEL
LIN {X 0,Y 212.139,Z 554.295,A -85,B 0,C 180,E1 -22730.656,E2 -22730.656} C_VEL
LIN {X 0,Y 207.541,Z 563.033,A -85,B 0,C 180,E1 -22731.039,E2 -22731.039} C_VEL
LIN {X 0,Y 202.621,Z 571.305,A -85,B 0,C 180,E1 -22731.589,E2 -22731.589} C_VEL
LIN {X 0,Y 200.366,Z 576.132,A -85,B 0,C 180,E1 -22732.241,E2 -22732.241} C_VEL
LIN {X 0,Y 196.423,Z 585.859,A -85,B 0,C 180,E1 -22734.135,E2 -22734.135} C_VEL
LIN {X 0,Y 191.521,Z 595.829,A -85,B 0,C 180,E1 -22736.604,E2 -22736.604} C_VEL
LIN {X 0,Y 186.696,Z 604.606,A -85,B 0,C 180,E1 -22739.458,E2 -22739.458} C_VEL
LIN {X 0,Y 182.557,Z 611.664,A -85,B 0,C 180,E1 -22742.487,E2 -22742.487} C_VEL
LIN {X 0,Y 178.905,Z 617.317,A -85,B 0,C 180,E1 -22745.641,E2 -22745.641} C_VEL
LIN {X 0,Y 175.705,Z 621.793,A -85,B 0,C 180,E1 -22748.902,E2 -22748.902} C_VEL
LIN {X 0,Y 173.892,Z 624.16,A -85,B 0,C 180,E1 -22751.137,E2 -22751.137} C_VEL
LIN {X 0,Y 171.248,Z 627.649,A -85,B 0,C 180,E1 -22755.746,E2 -22755.746} C_VEL
LIN {X 0,Y 170.318,Z 628.761,A -85,B 0,C 180,E1 -22758.094,E2 -22758.094} C_VEL
LIN {X 0,Y 169.177,Z 629.806,A -85,B 0,C 180,E1 -22762.842,E2 -22762.842} C_VEL
LIN {X 0,Y 168.938,Z 629.763,A -85,B 0,C 180,E1 -22765.228,E2 -22765.228} C_VEL
LIN {X 0,Y 168.839,Z 629.32,A -85,B 0,C 180,E1 -22767.615,E2 -22767.615} C_VEL
LIN {X 0,Y 168.91,Z 628.454,A -85,B 0,C 180,E1 -22770.001,E2 -22770.001} C_VEL
LIN {X 0,Y 168.819,Z 627.183,A -85,B 0,C 180,E1 -22772.386,E2 -22772.386} C_VEL
LIN {X 0,Y 168.965,Z 624.475,A -85,B 0,C 180,E1 -22775.969,E2 -22775.969} C_VEL
LIN {X 0,Y 169.433,Z 620.725,A -85,B 0,C 180,E1 -22779.551,E2 -22779.551} C_VEL
LIN {X 0,Y 170.369,Z 615.833,A -85,B 0,C 180,E1 -22783.114,E2 -22783.114} C_VEL
LIN {X 0,Y 171.811,Z 609.645,A -85,B 0,C 180,E1 -22786.639,E2 -22786.639} C_VEL
LIN {X 0,Y 173.851,Z 601.93,A -85,B 0,C 180,E1 -22790.098,E2 -22790.098} C_VEL
LIN {X 0,Y 175.981,Z 594.005,A -85,B 0,C 180,E1 -22792.916,E2 -22792.916} C_VEL
LIN {X 0,Y 178.359,Z 584.289,A -85,B 0,C 180,E1 -22795.686,E2 -22795.686} C_VEL
LIN {X 0,Y 180.895,Z 573.497,A -85,B 0,C 180,E1 -22798.104,E2 -22798.104} C_VEL
LIN {X 0,Y 183.227,Z 563.064,A -85,B 0,C 180,E1 -22799.91,E2 -22799.91} C_VEL
LIN {X 0,Y 185.252,Z 551.621,A -85,B 0,C 180,E1 -22801.442,E2 -22801.442} C_VEL
LIN {X 0,Y 187,Z 538.703,A -85,B 0,C 180,E1 -22802.701,E2 -22802.701} C_VEL
LIN {X 0,Y 188.354,Z 525.154,A -85,B 0,C 180,E1 -22803.552,E2 -22803.552} C_VEL
LIN {X 0,Y 190.777,Z 471.213,A -85,B 0,C 180,E1 -22805.506,E2 -22805.506} C_VEL
LIN {X 0,Y 189.37,Z 459.327,A -85,B 0,C 180,E1 -22806.272,E2 -22806.272} C_VEL
LIN {X 0,Y 184.284,Z 445.292,A -85,B 0,C 180,E1 -22807.856,E2 -22807.856} C_VEL
LIN {X 0,Y 178.266,Z 431.376,A -85,B 0,C 180,E1 -22809.756,E2 -22809.756} C_VEL
LIN {X 0,Y 173.054,Z 421.397,A -85,B 0,C 180,E1 -22811.439,E2 -22811.439} C_VEL
LIN {X 0,Y 171.578,Z 418.546,A -85,B 0,C 180,E1 -22812.028,E2 -22812.028} C_VEL
LIN {X 0,Y 171.409,Z 417.708,A -85,B 0,C 180,E1 -22812.584,E2 -22812.584} C_VEL
LIN {X 0,Y 171.441,Z 417.578,A -85,B 0,C 180,E1 -22817.551,E2 -22817.551} C_VEL
LIN {X 0,Y 171.437,Z 417.625,A -85,B 0,C 180,E1 -22822.054,E2 -22822.054} C_VEL
LIN {X 0,Y 171.418,Z 417.635,A -85,B 0,C 180,E1 -22827.792,E2 -22827.792} C_VEL
LIN {X 0,Y 171.447,Z 417.607,A -85,B 0,C 180,E1 -22830.534,E2 -22830.534} C_VEL
LIN {X 0,Y 171.444,Z 417.629,A -85,B 0,C 180,E1 -22835.799,E2 -22835.799} C_VEL
LIN {X 0,Y 171.576,Z 417.584,A -85,B 0,C 180,E1 -22840.871,E2 -22840.871} C_VEL
LIN {X 0,Y 171.574,Z 417.609,A -85,B 0,C 180,E1 -22845.772,E2 -22845.772} C_VEL
LIN {X 0,Y 171.847,Z 417.542,A -85,B 0,C 180,E1 -22850.585,E2 -22850.585} C_VEL
LIN {X 0,Y 171.814,Z 417.584,A -85,B 0,C 180,E1 -22855.307,E2 -22855.307} C_VEL
LIN {X 0,Y 172.331,Z 417.477,A -85,B 0,C 180,E1 -22860,E2 -22860} C_VEL
LIN {X 0,Y 171.815,Z 417.575,A -85,B 0,C 180,E1 -22864.692,E2 -22864.692} C_VEL
LIN {X 0,Y 171.849,Z 417.563,A -85,B 0,C 180,E1 -22869.415,E2 -22869.415} C_VEL
LIN {X 0,Y 171.573,Z 417.578,A -85,B 0,C 180,E1 -22874.227,E2 -22874.227} C_VEL
LIN {X 0,Y 171.544,Z 417.612,A -85,B 0,C 180,E1 -22879.562,E2 -22879.562} C_VEL
LIN {X 0,Y 171.461,Z 417.598,A -85,B 0,C 180,E1 -22885.611,E2 -22885.611} C_VEL
LIN {X 0,Y 171.458,Z 417.617,A -85,B 0,C 180,E1 -22890.596,E2 -22890.596} C_VEL
LIN {X 0,Y 171.392,Z 417.609,A -85,B 0,C 180,E1 -22895.035,E2 -22895.035} C_VEL
LIN {X 0,Y 171.357,Z 417.638,A -85,B 0,C 180,E1 -22898.808,E2 -22898.808} C_VEL
LIN {X 0,Y 171.344,Z 417.63,A -85,B 0,C 180,E1 -22904.209,E2 -22904.209} C_VEL
LIN {X 0,Y 171.38,Z 417.619,A -85,B 0,C 180,E1 -22908.995,E2 -22908.995} C_VEL
LIN {X 0,Y 171.436,Z 417.634,A -85,B 0,C 180,E1 -22912.054,E2 -22912.054} C_VEL
LIN {X 0,Y 171.42,Z 417.574,A -85,B 0,C 180,E1 -22917.793,E2 -22917.793} C_VEL
LIN {X 0,Y 171.519,Z 417.875,A -85,B 0,C 180,E1 -22920.973,E2 -22920.973} C_VEL
LIN {X 0,Y 171.754,Z 418.879,A -85,B 0,C 180,E1 -22921.35,E2 -22921.35} C_VEL
LIN {X 0,Y 173.413,Z 421.698,A -85,B 0,C 180,E1 -22921.917,E2 -22921.917} C_VEL
LIN {X 0,Y 181.463,Z 435.773,A -85,B 0,C 180,E1 -22924.39,E2 -22924.39} C_VEL
LIN {X 0,Y 187.103,Z 449.284,A -85,B 0,C 180,E1 -22926.122,E2 -22926.122} C_VEL
LIN {X 0,Y 191.11,Z 460.942,A -85,B 0,C 180,E1 -22927.364,E2 -22927.364} C_VEL
LIN {X 0,Y 190.581,Z 476.287,A -85,B 0,C 180,E1 -22927.934,E2 -22927.934} C_VEL
LIN {X 0,Y 188.368,Z 521.318,A -85,B 0,C 180,E1 -22929.558,E2 -22929.558} C_VEL
LIN {X 0,Y 187.032,Z 534.951,A -85,B 0,C 180,E1 -22930.451,E2 -22930.451} C_VEL
LIN {X 0,Y 185.181,Z 548.218,A -85,B 0,C 180,E1 -22931.78,E2 -22931.78} C_VEL
LIN {X 0,Y 183.03,Z 560.192,A -85,B 0,C 180,E1 -22933.463,E2 -22933.463} C_VEL
LIN {X 0,Y 180.414,Z 571.941,A -85,B 0,C 180,E1 -22935.621,E2 -22935.621} C_VEL
LIN {X 0,Y 178.239,Z 581.034,A -85,B 0,C 180,E1 -22937.764,E2 -22937.764} C_VEL
LIN {X 0,Y 175.987,Z 589.538,A -85,B 0,C 180,E1 -22940.228,E2 -22940.228} C_VEL
LIN {X 0,Y 174.038,Z 597.348,A -85,B 0,C 180,E1 -22943.041,E2 -22943.041} C_VEL
LIN {X 0,Y 171.93,Z 605.003,A -85,B 0,C 180,E1 -22946.484,E2 -22946.484} C_VEL
LIN {X 0,Y 170.48,Z 611.147,A -85,B 0,C 180,E1 -22949.999,E2 -22949.999} C_VEL
LIN {X 0,Y 169.573,Z 616.017,A -85,B 0,C 180,E1 -22953.564,E2 -22953.564} C_VEL
LIN {X 0,Y 168.899,Z 619.776,A -85,B 0,C 180,E1 -22957.17,E2 -22957.17} C_VEL
LIN {X 0,Y 168.575,Z 621.724,A -85,B 0,C 180,E1 -22959.599,E2 -22959.599} C_VEL
LIN {X 0,Y 168.452,Z 623.215,A -85,B 0,C 180,E1 -22962.04,E2 -22962.04} C_VEL
LIN {X 0,Y 168.693,Z 624.847,A -85,B 0,C 180,E1 -22966.622,E2 -22966.622} C_VEL
LIN {X 0,Y 169.047,Z 625.166,A -85,B 0,C 180,E1 -22969.425,E2 -22969.425} C_VEL
LIN {X 0,Y 169.603,Z 624.958,A -85,B 0,C 180,E1 -22971.896,E2 -22971.896} C_VEL
LIN {X 0,Y 170.662,Z 624.107,A -85,B 0,C 180,E1 -22975.045,E2 -22975.045} C_VEL
LIN {X 0,Y 172.751,Z 621.821,A -85,B 0,C 180,E1 -22979.221,E2 -22979.221} C_VEL
LIN {X 0,Y 175.066,Z 618.979,A -85,B 0,C 180,E1 -22982.537,E2 -22982.537} C_VEL
LIN {X 0,Y 178.352,Z 614.493,A -85,B 0,C 180,E1 -22986.232,E2 -22986.232} C_VEL
LIN {X 0,Y 182.391,Z 608.429,A -85,B 0,C 180,E1 -22989.869,E2 -22989.869} C_VEL
LIN {X 0,Y 186.32,Z 602.061,A -85,B 0,C 180,E1 -22992.761,E2 -22992.761} C_VEL
LIN {X 0,Y 190.959,Z 593.867,A -85,B 0,C 180,E1 -22995.632,E2 -22995.632} C_VEL
LIN {X 0,Y 195.667,Z 584.327,A -85,B 0,C 180,E1 -22998.183,E2 -22998.183} C_VEL
LIN {X 0,Y 199.943,Z 574.345,A -85,B 0,C 180,E1 -23000.254,E2 -23000.254} C_VEL
LIN {X 0,Y 204.079,Z 562.947,A -85,B 0,C 180,E1 -23002.074,E2 -23002.074} C_VEL
LIN {X 0,Y 207.54,Z 550.843,A -85,B 0,C 180,E1 -23003.536,E2 -23003.536} C_VEL
LIN {X 0,Y 210.508,Z 538.151,A -85,B 0,C 180,E1 -23004.61,E2 -23004.61} C_VEL
LIN {X 0,Y 212.499,Z 525.563,A -85,B 0,C 180,E1 -23005.352,E2 -23005.352} C_VEL
LIN {X 0,Y 213.924,Z 509.17,A -85,B 0,C 180,E1 -23005.925,E2 -23005.925} C_VEL
LIN {X 0,Y 215.513,Z 484.187,A -85,B 0,C 180,E1 -23006.703,E2 -23006.703} C_VEL
LIN {X 0,Y 210.196,Z 472.504,A -85,B 0,C 180,E1 -23009.047,E2 -23009.047} C_VEL
LIN {X 0,Y 204.573,Z 461.777,A -85,B 0,C 180,E1 -23011.724,E2 -23011.724} C_VEL
LIN {X 0,Y 198.776,Z 452.233,A -85,B 0,C 180,E1 -23014.777,E2 -23014.777} C_VEL
LIN {X 0,Y 195.913,Z 447.742,A -85,B 0,C 180,E1 -23016.449,E2 -23016.449} C_VEL
LIN {X 0,Y 193.29,Z 444.118,A -85,B 0,C 180,E1 -23018.066,E2 -23018.066} C_VEL
LIN {X 0,Y 190.422,Z 440.202,A -85,B 0,C 180,E1 -23019.986,E2 -23019.986} C_VEL
LIN {X 0,Y 187.236,Z 436.605,A -85,B 0,C 180,E1 -23022.286,E2 -23022.286} C_VEL
LIN {X 0,Y 186.133,Z 434.688,A -85,B 0,C 180,E1 -23023.215,E2 -23023.215} C_VEL
LIN {X 0,Y 183.531,Z 432.274,A -85,B 0,C 180,E1 -23025.379,E2 -23025.379} C_VEL
LIN {X 0,Y 181.783,Z 429.312,A -85,B 0,C 180,E1 -23027.156,E2 -23027.156} C_VEL
LIN {X 0,Y 179.364,Z 427.472,A -85,B 0,C 180,E1 -23029.706,E2 -23029.706} C_VEL
LIN {X 0,Y 177.779,Z 424.715,A -85,B 0,C 180,E1 -23031.904,E2 -23031.904} C_VEL
LIN {X 0,Y 177.368,Z 423.602,A -85,B 0,C 180,E1 -23032.601,E2 -23032.601} C_VEL
LIN {X 0,Y 174.65,Z 422.233,A -85,B 0,C 180,E1 -23037.117,E2 -23037.117} C_VEL
LIN {X 0,Y 173.413,Z 420.634,A -85,B 0,C 180,E1 -23040.581,E2 -23040.581} C_VEL
LIN {X 0,Y 172.619,Z 420.061,A -85,B 0,C 180,E1 -23044.671,E2 -23044.671} C_VEL
LIN {X 0,Y 172.628,Z 420.019,A -85,B 0,C 180,E1 -23048.192,E2 -23048.192} C_VEL
LIN {X 0,Y 173.331,Z 421.341,A -85,B 0,C 180,E1 -23052.291,E2 -23052.291} C_VEL
LIN {X 0,Y 177.088,Z 423.874,A -85,B 0,C 180,E1 -23059.931,E2 -23059.931} C_VEL
LIN {X 0,Y 178.5,Z 426.826,A -85,B 0,C 180,E1 -23062.117,E2 -23062.117} C_VEL
LIN {X 0,Y 180.952,Z 429.034,A -85,B 0,C 180,E1 -23064.917,E2 -23064.917} C_VEL
LIN {X 0,Y 182.197,Z 430.232,A -85,B 0,C 180,E1 -23066.161,E2 -23066.161} C_VEL
LIN {X 0,Y 184.364,Z 433.381,A -85,B 0,C 180,E1 -23068.227,E2 -23068.227} C_VEL
LIN {X 0,Y 187.351,Z 437.014,A -85,B 0,C 180,E1 -23070.678,E2 -23070.678} C_VEL
LIN {X 0,Y 190.433,Z 441.389,A -85,B 0,C 180,E1 -23072.97,E2 -23072.97} C_VEL
LIN {X 0,Y 194.99,Z 448.207,A -85,B 0,C 180,E1 -23075.975,E2 -23075.975} C_VEL
LIN {X 0,Y 198.827,Z 454.535,A -85,B 0,C 180,E1 -23078.253,E2 -23078.253} C_VEL
LIN {X 0,Y 203.832,Z 463.308,A -85,B 0,C 180,E1 -23080.928,E2 -23080.928} C_VEL
LIN {X 0,Y 208.944,Z 473.158,A -85,B 0,C 180,E1 -23083.406,E2 -23083.406} C_VEL
LIN {X 0,Y 213.644,Z 483.674,A -85,B 0,C 180,E1 -23085.537,E2 -23085.537} C_VEL
LIN {X 0,Y 215.428,Z 488.329,A -85,B 0,C 180,E1 -23086.332,E2 -23086.332} C_VEL
LIN {X 0,Y 212.694,Z 526.254,A -85,B 0,C 180,E1 -23087.499,E2 -23087.499} C_VEL
LIN {X 0,Y 210.652,Z 540.088,A -85,B 0,C 180,E1 -23088.226,E2 -23088.226} C_VEL
LIN {X 0,Y 207.896,Z 552.804,A -85,B 0,C 180,E1 -23089.244,E2 -23089.244} C_VEL
LIN {X 0,Y 204.417,Z 564.477,A -85,B 0,C 180,E1 -23090.504,E2 -23090.504} C_VEL
LIN {X 0,Y 200.517,Z 575.71,A -85,B 0,C 180,E1 -23092.168,E2 -23092.168} C_VEL
LIN {X 0,Y 200.366,Z 576.132,A -85,B 0,C 180,E1 -23092.241,E2 -23092.241} C_VEL
LIN {X 0,Y 198.048,Z 580.914,A -85,B 0,C 180,E1 -23092.984,E2 -23092.984} C_VEL
LIN {X 0,Y 192.582,Z 588.401,A -85,B 0,C 180,E1 -23094.02,E2 -23094.02} C_VEL
LIN {X 0,Y 186.784,Z 595.356,A -85,B 0,C 180,E1 -23095.252,E2 -23095.252} C_VEL
LIN {X 0,Y 183.996,Z 599.304,A -85,B 0,C 180,E1 -23096.306,E2 -23096.306} C_VEL
LIN {X 0,Y 179.085,Z 607.485,A -85,B 0,C 180,E1 -23099.326,E2 -23099.326} C_VEL
LIN {X 0,Y 174.973,Z 613.957,A -85,B 0,C 180,E1 -23102.491,E2 -23102.491} C_VEL
LIN {X 0,Y 171.273,Z 619.133,A -85,B 0,C 180,E1 -23105.775,E2 -23105.775} C_VEL
LIN {X 0,Y 168.129,Z 623.168,A -85,B 0,C 180,E1 -23109.189,E2 -23109.189} C_VEL
LIN {X 0,Y 165.615,Z 626.177,A -85,B 0,C 180,E1 -23112.72,E2 -23112.72} C_VEL
LIN {X 0,Y 164.36,Z 627.675,A -85,B 0,C 180,E1 -23115.135,E2 -23115.135} C_VEL
LIN {X 0,Y 162.616,Z 629.417,A -85,B 0,C 180,E1 -23120.046,E2 -23120.046} C_VEL
LIN {X 0,Y 161.858,Z 629.645,A -85,B 0,C 180,E1 -23125.019,E2 -23125.019} C_VEL
LIN {X 0,Y 161.733,Z 628.956,A -85,B 0,C 180,E1 -23128.111,E2 -23128.111} C_VEL
LIN {X 0,Y 161.822,Z 628.249,A -85,B 0,C 180,E1 -23130.001,E2 -23130.001} C_VEL
LIN {X 0,Y 161.721,Z 626.947,A -85,B 0,C 180,E1 -23132.491,E2 -23132.491} C_VEL
LIN {X 0,Y 161.89,Z 624.175,A -85,B 0,C 180,E1 -23136.231,E2 -23136.231} C_VEL
LIN {X 0,Y 162.413,Z 620.357,A -85,B 0,C 180,E1 -23139.968,E2 -23139.968} C_VEL
LIN {X 0,Y 163.42,Z 615.391,A -85,B 0,C 180,E1 -23143.682,E2 -23143.682} C_VEL
LIN {X 0,Y 165.004,Z 609.126,A -85,B 0,C 180,E1 -23147.347,E2 -23147.347} C_VEL
LIN {X 0,Y 167.156,Z 601.275,A -85,B 0,C 180,E1 -23150.94,E2 -23150.94} C_VEL
LIN {X 0,Y 169.146,Z 594.255,A -85,B 0,C 180,E1 -23153.528,E2 -23153.528} C_VEL
LIN {X 0,Y 171.657,Z 584.461,A -85,B 0,C 180,E1 -23156.439,E2 -23156.439} C_VEL
LIN {X 0,Y 174.289,Z 573.722,A -85,B 0,C 180,E1 -23158.94,E2 -23158.94} C_VEL
LIN {X 0,Y 176.704,Z 563.361,A -85,B 0,C 180,E1 -23160.802,E2 -23160.802} C_VEL
LIN {X 0,Y 178.981,Z 550.939,A -85,B 0,C 180,E1 -23162.511,E2 -23162.511} C_VEL
LIN {X 0,Y 180.84,Z 537.829,A -85,B 0,C 180,E1 -23163.795,E2 -23163.795} C_VEL
LIN {X 0,Y 182.134,Z 525.027,A -85,B 0,C 180,E1 -23164.607,E2 -23164.607} C_VEL
LIN {X 0,Y 184.637,Z 471.698,A -85,B 0,C 180,E1 -23166.591,E2 -23166.591} C_VEL
LIN {X 0,Y 183.352,Z 461.215,A -85,B 0,C 180,E1 -23167.31,E2 -23167.31} C_VEL
LIN {X 0,Y 177.331,Z 444.923,A -85,B 0,C 180,E1 -23169.304,E2 -23169.304} C_VEL
LIN {X 0,Y 171.552,Z 432.031,A -85,B 0,C 180,E1 -23171.258,E2 -23171.258} C_VEL
LIN {X 0,Y 168.117,Z 425.685,A -85,B 0,C 180,E1 -23172.429,E2 -23172.429} C_VEL
LIN {X 0,Y 166.104,Z 422.381,A -85,B 0,C 180,E1 -23173.125,E2 -23173.125} C_VEL
LIN {X 0,Y 164.542,Z 419.48,A -85,B 0,C 180,E1 -23173.77,E2 -23173.77} C_VEL
LIN {X 0,Y 164.373,Z 418.562,A -85,B 0,C 180,E1 -23174.367,E2 -23174.367} C_VEL
LIN {X 0,Y 164.375,Z 418.45,A -85,B 0,C 180,E1 -23176.835,E2 -23176.835} C_VEL
LIN {X 0,Y 164.371,Z 418.505,A -85,B 0,C 180,E1 -23180.32,E2 -23180.32} C_VEL
LIN {X 0,Y 164.331,Z 418.509,A -85,B 0,C 180,E1 -23186.222,E2 -23186.222} C_VEL
LIN {X 0,Y 164.389,Z 418.497,A -85,B 0,C 180,E1 -23189.134,E2 -23189.134} C_VEL
LIN {X 0,Y 164.405,Z 418.506,A -85,B 0,C 180,E1 -23194.692,E2 -23194.692} C_VEL
LIN {X 0,Y 164.484,Z 418.463,A -85,B 0,C 180,E1 -23200.051,E2 -23200.051} C_VEL
LIN {X 0,Y 164.522,Z 418.49,A -85,B 0,C 180,E1 -23205.149,E2 -23205.149} C_VEL
LIN {X 0,Y 164.766,Z 418.421,A -85,B 0,C 180,E1 -23210.176,E2 -23210.176} C_VEL
LIN {X 0,Y 164.83,Z 418.436,A -85,B 0,C 180,E1 -23212.651,E2 -23212.651} C_VEL
LIN {X 0,Y 165.046,Z 418.412,A -85,B 0,C 180,E1 -23217.559,E2 -23217.559} C_VEL
LIN {X 0,Y 165.293,Z 418.352,A -85,B 0,C 180,E1 -23220,E2 -23220} C_VEL
LIN {X 0,Y 164.764,Z 418.454,A -85,B 0,C 180,E1 -23224.894,E2 -23224.894} C_VEL
LIN {X 0,Y 164.833,Z 418.451,A -85,B 0,C 180,E1 -23227.349,E2 -23227.349} C_VEL
LIN {X 0,Y 164.702,Z 418.429,A -85,B 0,C 180,E1 -23231.061,E2 -23231.061} C_VEL
LIN {X 0,Y 164.483,Z 418.494,A -85,B 0,C 180,E1 -23237.403,E2 -23237.403} C_VEL
LIN {X 0,Y 164.473,Z 418.489,A -85,B 0,C 180,E1 -23239.989,E2 -23239.989} C_VEL
LIN {X 0,Y 164.388,Z 418.484,A -85,B 0,C 180,E1 -23246.13,E2 -23246.13} C_VEL
LIN {X 0,Y 164.388,Z 418.49,A -85,B 0,C 180,E1 -23251.235,E2 -23251.235} C_VEL
LIN {X 0,Y 164.294,Z 418.514,A -85,B 0,C 180,E1 -23256.789,E2 -23256.789} C_VEL
LIN {X 0,Y 164.292,Z 418.507,A -85,B 0,C 180,E1 -23259.916,E2 -23259.916} C_VEL
LIN {X 0,Y 164.279,Z 418.499,A -85,B 0,C 180,E1 -23263.342,E2 -23263.342} C_VEL
LIN {X 0,Y 164.321,Z 418.512,A -85,B 0,C 180,E1 -23266.818,E2 -23266.818} C_VEL
LIN {X 0,Y 164.344,Z 418.5,A -85,B 0,C 180,E1 -23270.331,E2 -23270.331} C_VEL
LIN {X 0,Y 164.344,Z 418.481,A -85,B 0,C 180,E1 -23274.342,E2 -23274.342} C_VEL
LIN {X 0,Y 164.428,Z 418.719,A -85,B 0,C 180,E1 -23279.143,E2 -23279.143} C_VEL
LIN {X 0,Y 164.68,Z 419.742,A -85,B 0,C 180,E1 -23279.576,E2 -23279.576} C_VEL
LIN {X 0,Y 166.324,Z 422.523,A -85,B 0,C 180,E1 -23280.195,E2 -23280.195} C_VEL
LIN {X 0,Y 174.418,Z 436.134,A -85,B 0,C 180,E1 -23282.874,E2 -23282.874} C_VEL
LIN {X 0,Y 178.165,Z 443.892,A -85,B 0,C 180,E1 -23284.081,E2 -23284.081} C_VEL
LIN {X 0,Y 183.94,Z 459.279,A -85,B 0,C 180,E1 -23285.971,E2 -23285.971} C_VEL
LIN {X 0,Y 185.051,Z 462.718,A -85,B 0,C 180,E1 -23286.338,E2 -23286.338} C_VEL
LIN {X 0,Y 182.189,Z 520.75,A -85,B 0,C 180,E1 -23288.47,E2 -23288.47} C_VEL
LIN {X 0,Y 180.81,Z 534.459,A -85,B 0,C 180,E1 -23289.371,E2 -23289.371} C_VEL
LIN {X 0,Y 179.025,Z 546.856,A -85,B 0,C 180,E1 -23290.608,E2 -23290.608} C_VEL
LIN {X 0,Y 177.037,Z 558.319,A -85,B 0,C 180,E1 -23292.197,E2 -23292.197} C_VEL
LIN {X 0,Y 174.496,Z 569.544,A -85,B 0,C 180,E1 -23294.225,E2 -23294.225} C_VEL
LIN {X 0,Y 172.032,Z 579.091,A -85,B 0,C 180,E1 -23296.414,E2 -23296.414} C_VEL
LIN {X 0,Y 169.469,Z 588.818,A -85,B 0,C 180,E1 -23299.244,E2 -23299.244} C_VEL
LIN {X 0,Y 167.344,Z 596.781,A -85,B 0,C 180,E1 -23302.155,E2 -23302.155} C_VEL
LIN {X 0,Y 165.13,Z 604.59,A -85,B 0,C 180,E1 -23305.728,E2 -23305.728} C_VEL
LIN {X 0,Y 163.82,Z 609.905,A -85,B 0,C 180,E1 -23308.77,E2 -23308.77} C_VEL
LIN {X 0,Y 162.706,Z 615.068,A -85,B 0,C 180,E1 -23312.475,E2 -23312.475} C_VEL
LIN {X 0,Y 161.964,Z 619.085,A -85,B 0,C 180,E1 -23316.227,E2 -23316.227} C_VEL
LIN {X 0,Y 161.434,Z 622.063,A -85,B 0,C 180,E1 -23320.028,E2 -23320.028} C_VEL
LIN {X 0,Y 161.359,Z 623.473,A -85,B 0,C 180,E1 -23322.578,E2 -23322.578} C_VEL
LIN {X 0,Y 161.646,Z 624.938,A -85,B 0,C 180,E1 -23326.96,E2 -23326.96} C_VEL
LIN {X 0,Y 162.091,Z 625.257,A -85,B 0,C 180,E1 -23330.295,E2 -23330.295} C_VEL
LIN {X 0,Y 162.748,Z 624.994,A -85,B 0,C 180,E1 -23332.869,E2 -23332.869} C_VEL
LIN {X 0,Y 163.772,Z 624.245,A -85,B 0,C 180,E1 -23335.687,E2 -23335.687} C_VEL
LIN {X 0,Y 164.837,Z 623.244,A -85,B 0,C 180,E1 -23337.968,E2 -23337.968} C_VEL
LIN {X 0,Y 167.146,Z 620.752,A -85,B 0,C 180,E1 -23341.706,E2 -23341.706} C_VEL
LIN {X 0,Y 170.104,Z 617.193,A -85,B 0,C 180,E1 -23345.338,E2 -23345.338} C_VEL
LIN {X 0,Y 173.685,Z 612.448,A -85,B 0,C 180,E1 -23348.842,E2 -23348.842} C_VEL
LIN {X 0,Y 177.824,Z 606.359,A -85,B 0,C 180,E1 -23352.21,E2 -23352.21} C_VEL
LIN {X 0,Y 182.64,Z 598.723,A -85,B 0,C 180,E1 -23355.386,E2 -23355.386} C_VEL
LIN {X 0,Y 187.172,Z 590.668,A -85,B 0,C 180,E1 -23357.966,E2 -23357.966} C_VEL
LIN {X 0,Y 191.8,Z 581.277,A -85,B 0,C 180,E1 -23360.306,E2 -23360.306} C_VEL
LIN {X 0,Y 195.859,Z 571.839,A -85,B 0,C 180,E1 -23362.129,E2 -23362.129} C_VEL
LIN {X 0,Y 200,Z 560.05,A -85,B 0,C 180,E1 -23363.92,E2 -23363.92} C_VEL
LIN {X 0,Y 203.29,Z 548.772,A -85,B 0,C 180,E1 -23365.189,E2 -23365.189} C_VEL
LIN {X 0,Y 206.19,Z 535.723,A -85,B 0,C 180,E1 -23366.236,E2 -23366.236} C_VEL
LIN {X 0,Y 208.274,Z 522.085,A -85,B 0,C 180,E1 -23366.942,E2 -23366.942} C_VEL
LIN {X 0,Y 210.779,Z 486.842,A -85,B 0,C 180,E1 -23368.076,E2 -23368.076} C_VEL
LIN {X 0,Y 205.765,Z 475.681,A -85,B 0,C 180,E1 -23370.454,E2 -23370.454} C_VEL
LIN {X 0,Y 200.966,Z 466.455,A -85,B 0,C 180,E1 -23372.898,E2 -23372.898} C_VEL
LIN {X 0,Y 195.448,Z 457.006,A -85,B 0,C 180,E1 -23376.017,E2 -23376.017} C_VEL
LIN {X 0,Y 192.743,Z 452.868,A -85,B 0,C 180,E1 -23377.692,E2 -23377.692} C_VEL
LIN {X 0,Y 190.722,Z 450.037,A -85,B 0,C 180,E1 -23379.015,E2 -23379.015} C_VEL
LIN {X 0,Y 187.738,Z 445.959,A -85,B 0,C 180,E1 -23381.129,E2 -23381.129} C_VEL
LIN {X 0,Y 184.903,Z 442.406,A -85,B 0,C 180,E1 -23383.34,E2 -23383.34} C_VEL
LIN {X 0,Y 183.863,Z 440.971,A -85,B 0,C 180,E1 -23384.232,E2 -23384.232} C_VEL
LIN {X 0,Y 181.32,Z 438.105,A -85,B 0,C 180,E1 -23386.552,E2 -23386.552} C_VEL
LIN {X 0,Y 180.354,Z 436.185,A -85,B 0,C 180,E1 -23387.624,E2 -23387.624} C_VEL
LIN {X 0,Y 177.785,Z 433.969,A -85,B 0,C 180,E1 -23390.5,E2 -23390.5} C_VEL
LIN {X 0,Y 176.253,Z 431.069,A -85,B 0,C 180,E1 -23392.806,E2 -23392.806} C_VEL
LIN {X 0,Y 176.084,Z 430.538,A -85,B 0,C 180,E1 -23393.123,E2 -23393.123} C_VEL
LIN {X 0,Y 173.634,Z 429.19,A -85,B 0,C 180,E1 -23397.39,E2 -23397.39} C_VEL
LIN {X 0,Y 172.368,Z 427.545,A -85,B 0,C 180,E1 -23401.168,E2 -23401.168} C_VEL
LIN {X 0,Y 171.69,Z 426.878,A -85,B 0,C 180,E1 -23407.054,E2 -23407.054} C_VEL
LIN {X 0,Y 172.108,Z 427.839,A -85,B 0,C 180,E1 -23410.836,E2 -23410.836} C_VEL
LIN {X 0,Y 175.772,Z 430.77,A -85,B 0,C 180,E1 -23419.342,E2 -23419.342} C_VEL
LIN {X 0,Y 177.416,Z 433.956,A -85,B 0,C 180,E1 -23421.934,E2 -23421.934} C_VEL
LIN {X 0,Y 180.447,Z 436.649,A -85,B 0,C 180,E1 -23425.368,E2 -23425.368} C_VEL
LIN {X 0,Y 182.681,Z 439.996,A -85,B 0,C 180,E1 -23427.618,E2 -23427.618} C_VEL
LIN {X 0,Y 185.25,Z 443.232,A -85,B 0,C 180,E1 -23429.833,E2 -23429.833} C_VEL
LIN {X 0,Y 189.301,Z 449.294,A -85,B 0,C 180,E1 -23432.956,E2 -23432.956} C_VEL
LIN {X 0,Y 192.708,Z 454.662,A -85,B 0,C 180,E1 -23435.277,E2 -23435.277} C_VEL
LIN {X 0,Y 195.969,Z 460.145,A -85,B 0,C 180,E1 -23437.307,E2 -23437.307} C_VEL
LIN {X 0,Y 201.605,Z 470.386,A -85,B 0,C 180,E1 -23440.466,E2 -23440.466} C_VEL
LIN {X 0,Y 206.879,Z 481.406,A -85,B 0,C 180,E1 -23443.132,E2 -23443.132} C_VEL
LIN {X 0,Y 210.689,Z 490.676,A -85,B 0,C 180,E1 -23444.95,E2 -23444.95} C_VEL
LIN {X 0,Y 208.043,Z 525.765,A -85,B 0,C 180,E1 -23446.025,E2 -23446.025} C_VEL
LIN {X 0,Y 205.977,Z 539.481,A -85,B 0,C 180,E1 -23446.738,E2 -23446.738} C_VEL
LIN {X 0,Y 203.197,Z 552.232,A -85,B 0,C 180,E1 -23447.758,E2 -23447.758} C_VEL
LIN {X 0,Y 199.571,Z 564.014,A -85,B 0,C 180,E1 -23449.015,E2 -23449.015} C_VEL
LIN {X 0,Y 195.483,Z 575.319,A -85,B 0,C 180,E1 -23450.682,E2 -23450.682} C_VEL
LIN {X 0,Y 191.193,Z 585.526,A -85,B 0,C 180,E1 -23452.663,E2 -23452.663} C_VEL
LIN {X 0,Y 186.585,Z 594.733,A -85,B 0,C 180,E1 -23454.943,E2 -23454.943} C_VEL
LIN {X 0,Y 183.996,Z 599.304,A -85,B 0,C 180,E1 -23456.306,E2 -23456.306} C_VEL
LIN {X 0,Y 181.222,Z 603.08,A -85,B 0,C 180,E1 -23457.453,E2 -23457.453} C_VEL
LIN {X 0,Y 175.323,Z 608.801,A -85,B 0,C 180,E1 -23459.237,E2 -23459.237} C_VEL
LIN {X 0,Y 169.511,Z 613.867,A -85,B 0,C 180,E1 -23461.288,E2 -23461.288} C_VEL
LIN {X 0,Y 166.935,Z 616.571,A -85,B 0,C 180,E1 -23462.836,E2 -23462.836} C_VEL
LIN {X 0,Y 163.666,Z 620.749,A -85,B 0,C 180,E1 -23465.926,E2 -23465.926} C_VEL
LIN {X 0,Y 160.522,Z 624.368,A -85,B 0,C 180,E1 -23469.498,E2 -23469.498} C_VEL
LIN {X 0,Y 158.822,Z 626.248,A -85,B 0,C 180,E1 -23471.957,E2 -23471.957} C_VEL
LIN {X 0,Y 157.499,Z 627.685,A -85,B 0,C 180,E1 -23474.471,E2 -23474.471} C_VEL
LIN {X 0,Y 155.62,Z 629.362,A -85,B 0,C 180,E1 -23479.594,E2 -23479.594} C_VEL
LIN {X 0,Y 155.076,Z 629.635,A -85,B 0,C 180,E1 -23482.187,E2 -23482.187} C_VEL
LIN {X 0,Y 154.791,Z 629.511,A -85,B 0,C 180,E1 -23484.791,E2 -23484.791} C_VEL
LIN {X 0,Y 154.65,Z 628.536,A -85,B 0,C 180,E1 -23488.815,E2 -23488.815} C_VEL
LIN {X 0,Y 154.633,Z 626.708,A -85,B 0,C 180,E1 -23492.606,E2 -23492.606} C_VEL
LIN {X 0,Y 154.808,Z 623.869,A -85,B 0,C 180,E1 -23496.517,E2 -23496.517} C_VEL
LIN {X 0,Y 155.416,Z 619.983,A -85,B 0,C 180,E1 -23500.422,E2 -23500.422} C_VEL
LIN {X 0,Y 156.495,Z 614.942,A -85,B 0,C 180,E1 -23504.3,E2 -23504.3} C_VEL
LIN {X 0,Y 158.229,Z 608.59,A -85,B 0,C 180,E1 -23508.115,E2 -23508.115} C_VEL
LIN {X 0,Y 160.516,Z 600.599,A -85,B 0,C 180,E1 -23511.849,E2 -23511.849} C_VEL
LIN {X 0,Y 162.603,Z 593.242,A -85,B 0,C 180,E1 -23514.617,E2 -23514.617} C_VEL
LIN {X 0,Y 165.256,Z 583.525,A -85,B 0,C 180,E1 -23517.548,E2 -23517.548} C_VEL
LIN {X 0,Y 168.016,Z 572.605,A -85,B 0,C 180,E1 -23520.129,E2 -23520.129} C_VEL
LIN {X 0,Y 170.61,Z 561.969,A -85,B 0,C 180,E1 -23522.03,E2 -23522.03} C_VEL
LIN {X 0,Y 173.02,Z 549.092,A -85,B 0,C 180,E1 -23523.778,E2 -23523.778} C_VEL
LIN {X 0,Y 174.853,Z 536.114,A -85,B 0,C 180,E1 -23525.03,E2 -23525.03} C_VEL
LIN {X 0,Y 176.069,Z 523.326,A -85,B 0,C 180,E1 -23525.803,E2 -23525.803} C_VEL
LIN {X 0,Y 178.564,Z 472.445,A -85,B 0,C 180,E1 -23527.735,E2 -23527.735} C_VEL
LIN {X 0,Y 177.419,Z 463.167,A -85,B 0,C 180,E1 -23528.41,E2 -23528.41} C_VEL
LIN {X 0,Y 171.412,Z 446.93,A -85,B 0,C 180,E1 -23530.534,E2 -23530.534} C_VEL
LIN {X 0,Y 165.818,Z 434.545,A -85,B 0,C 180,E1 -23532.548,E2 -23532.548} C_VEL
LIN {X 0,Y 161.897,Z 427.516,A -85,B 0,C 180,E1 -23533.983,E2 -23533.983} C_VEL
LIN {X 0,Y 158.977,Z 423.048,A -85,B 0,C 180,E1 -23535.073,E2 -23535.073} C_VEL
LIN {X 0,Y 157.53,Z 420.376,A -85,B 0,C 180,E1 -23535.73,E2 -23535.73} C_VEL
LIN {X 0,Y 157.332,Z 419.46,A -85,B 0,C 180,E1 -23536.369,E2 -23536.369} C_VEL
LIN {X 0,Y 157.281,Z 419.395,A -85,B 0,C 180,E1 -23541.275,E2 -23541.275} C_VEL
LIN {X 0,Y 157.291,Z 419.372,A -85,B 0,C 180,E1 -23544.489,E2 -23544.489} C_VEL
LIN {X 0,Y 157.293,Z 419.394,A -85,B 0,C 180,E1 -23548.096,E2 -23548.096} C_VEL
LIN {X 0,Y 157.313,Z 419.377,A -85,B 0,C 180,E1 -23553.464,E2 -23553.464} C_VEL
LIN {X 0,Y 157.391,Z 419.345,A -85,B 0,C 180,E1 -23559.67,E2 -23559.67} C_VEL
LIN {X 0,Y 157.452,Z 419.372,A -85,B 0,C 180,E1 -23564.465,E2 -23564.465} C_VEL
LIN {X 0,Y 157.688,Z 419.3,A -85,B 0,C 180,E1 -23569.73,E2 -23569.73} C_VEL
LIN {X 0,Y 157.766,Z 419.31,A -85,B 0,C 180,E1 -23572.32,E2 -23572.32} C_VEL
LIN {X 0,Y 158.256,Z 419.227,A -85,B 0,C 180,E1 -23580,E2 -23580} C_VEL
LIN {X 0,Y 157.769,Z 419.33,A -85,B 0,C 180,E1 -23587.68,E2 -23587.68} C_VEL
LIN {X 0,Y 157.633,Z 419.306,A -85,B 0,C 180,E1 -23591.231,E2 -23591.231} C_VEL
LIN {X 0,Y 157.44,Z 419.352,A -85,B 0,C 180,E1 -23595.535,E2 -23595.535} C_VEL
LIN {X 0,Y 157.369,Z 419.361,A -85,B 0,C 180,E1 -23600.933,E2 -23600.933} C_VEL
LIN {X 0,Y 157.31,Z 419.371,A -85,B 0,C 180,E1 -23606.682,E2 -23606.682} C_VEL
LIN {X 0,Y 157.281,Z 419.361,A -85,B 0,C 180,E1 -23612.426,E2 -23612.426} C_VEL
LIN {X 0,Y 157.267,Z 419.382,A -85,B 0,C 180,E1 -23616.449,E2 -23616.449} C_VEL
LIN {X 0,Y 157.211,Z 419.374,A -85,B 0,C 180,E1 -23622.111,E2 -23622.111} C_VEL
LIN {X 0,Y 157.241,Z 419.383,A -85,B 0,C 180,E1 -23627.899,E2 -23627.899} C_VEL
LIN {X 0,Y 157.322,Z 419.369,A -85,B 0,C 180,E1 -23633.524,E2 -23633.524} C_VEL
LIN {X 0,Y 157.297,Z 419.527,A -85,B 0,C 180,E1 -23637.007,E2 -23637.007} C_VEL
LIN {X 0,Y 157.504,Z 420.492,A -85,B 0,C 180,E1 -23637.542,E2 -23637.542} C_VEL
LIN {X 0,Y 159.117,Z 423.321,A -85,B 0,C 180,E1 -23638.239,E2 -23638.239} C_VEL
LIN {X 0,Y 160.225,Z 424.808,A -85,B 0,C 180,E1 -23638.645,E2 -23638.645} C_VEL
LIN {X 0,Y 167.006,Z 436.065,A -85,B 0,C 180,E1 -23641.09,E2 -23641.09} C_VEL
LIN {X 0,Y 171.711,Z 444.828,A -85,B 0,C 180,E1 -23642.684,E2 -23642.684} C_VEL
LIN {X 0,Y 177.622,Z 460.181,A -85,B 0,C 180,E1 -23644.746,E2 -23644.746} C_VEL
LIN {X 0,Y 179.007,Z 464.772,A -85,B 0,C 180,E1 -23645.249,E2 -23645.249} C_VEL
LIN {X 0,Y 175.937,Z 521.916,A -85,B 0,C 180,E1 -23647.405,E2 -23647.405} C_VEL
LIN {X 0,Y 174.481,Z 535.731,A -85,B 0,C 180,E1 -23648.377,E2 -23648.377} C_VEL
LIN {X 0,Y 172.513,Z 548.521,A -85,B 0,C 180,E1 -23649.741,E2 -23649.741} C_VEL
LIN {X 0,Y 170.4,Z 559.506,A -85,B 0,C 180,E1 -23651.358,E2 -23651.358} C_VEL
LIN {X 0,Y 167.609,Z 571.036,A -85,B 0,C 180,E1 -23653.558,E2 -23653.558} C_VEL
LIN {X 0,Y 165.177,Z 580.325,A -85,B 0,C 180,E1 -23655.838,E2 -23655.838} C_VEL
LIN {X 0,Y 162.473,Z 589.867,A -85,B 0,C 180,E1 -23658.775,E2 -23658.775} C_VEL
LIN {X 0,Y 159.877,Z 599.023,A -85,B 0,C 180,E1 -23662.421,E2 -23662.421} C_VEL
LIN {X 0,Y 157.749,Z 606.409,A -85,B 0,C 180,E1 -23666.168,E2 -23666.168} C_VEL
LIN {X 0,Y 156.197,Z 612.331,A -85,B 0,C 180,E1 -23669.999,E2 -23669.999} C_VEL
LIN {X 0,Y 155.246,Z 617.234,A -85,B 0,C 180,E1 -23674.12,E2 -23674.12} C_VEL
LIN {X 0,Y 154.567,Z 620.565,A -85,B 0,C 180,E1 -23677.839,E2 -23677.839} C_VEL
LIN {X 0,Y 154.318,Z 622.366,A -85,B 0,C 180,E1 -23680.495,E2 -23680.495} C_VEL
LIN {X 0,Y 154.284,Z 623.729,A -85,B 0,C 180,E1 -23683.164,E2 -23683.164} C_VEL
LIN {X 0,Y 154.588,Z 625.024,A -85,B 0,C 180,E1 -23687.308,E2 -23687.308} C_VEL
LIN {X 0,Y 155.192,Z 625.338,A -85,B 0,C 180,E1 -23691.239,E2 -23691.239} C_VEL
LIN {X 0,Y 156.907,Z 624.383,A -85,B 0,C 180,E1 -23696.387,E2 -23696.387} C_VEL
LIN {X 0,Y 158.306,Z 623.15,A -85,B 0,C 180,E1 -23699.231,E2 -23699.231} C_VEL
LIN {X 0,Y 160.863,Z 620.567,A -85,B 0,C 180,E1 -23703.1,E2 -23703.1} C_VEL
LIN {X 0,Y 164.09,Z 616.904,A -85,B 0,C 180,E1 -23706.841,E2 -23706.841} C_VEL
LIN {X 0,Y 167.93,Z 612.044,A -85,B 0,C 180,E1 -23710.441,E2 -23710.441} C_VEL
LIN {X 0,Y 172.437,Z 605.843,A -85,B 0,C 180,E1 -23713.856,E2 -23713.856} C_VEL
LIN {X 0,Y 177.534,Z 598.077,A -85,B 0,C 180,E1 -23717.082,E2 -23717.082} C_VEL
LIN {X 0,Y 182.621,Z 589.249,A -85,B 0,C 180,E1 -23719.85,E2 -23719.85} C_VEL
LIN {X 0,Y 187.689,Z 579.103,A -85,B 0,C 180,E1 -23722.279,E2 -23722.279} C_VEL
LIN {X 0,Y 192.216,Z 568.584,A -85,B 0,C 180,E1 -23724.196,E2 -23724.196} C_VEL
LIN {X 0,Y 196.304,Z 556.593,A -85,B 0,C 180,E1 -23725.882,E2 -23725.882} C_VEL
LIN {X 0,Y 199.791,Z 544.193,A -85,B 0,C 180,E1 -23727.121,E2 -23727.121} C_VEL
LIN {X 0,Y 202.391,Z 531.529,A -85,B 0,C 180,E1 -23728.016,E2 -23728.016} C_VEL
LIN {X 0,Y 204.176,Z 517.914,A -85,B 0,C 180,E1 -23728.612,E2 -23728.612} C_VEL
LIN {X 0,Y 206.222,Z 489.586,A -85,B 0,C 180,E1 -23729.496,E2 -23729.496} C_VEL
LIN {X 0,Y 201.19,Z 478.322,A -85,B 0,C 180,E1 -23732.067,E2 -23732.067} C_VEL
LIN {X 0,Y 196.178,Z 468.691,A -85,B 0,C 180,E1 -23734.856,E2 -23734.856} C_VEL
LIN {X 0,Y 190.909,Z 459.702,A -85,B 0,C 180,E1 -23738.151,E2 -23738.151} C_VEL
LIN {X 0,Y 188.211,Z 455.932,A -85,B 0,C 180,E1 -23739.989,E2 -23739.989} C_VEL
LIN {X 0,Y 185.53,Z 452.179,A -85,B 0,C 180,E1 -23741.997,E2 -23741.997} C_VEL
LIN {X 0,Y 182.679,Z 448.277,A -85,B 0,C 180,E1 -23744.377,E2 -23744.377} C_VEL
LIN {X 0,Y 179.439,Z 444.284,A -85,B 0,C 180,E1 -23747.488,E2 -23747.488} C_VEL
LIN {X 0,Y 178.732,Z 442.876,A -85,B 0,C 180,E1 -23748.316,E2 -23748.316} C_VEL
LIN {X 0,Y 176.326,Z 440.595,A -85,B 0,C 180,E1 -23751.188,E2 -23751.188} C_VEL
LIN {X 0,Y 174.807,Z 437.526,A -85,B 0,C 180,E1 -23753.652,E2 -23753.652} C_VEL
LIN {X 0,Y 172.332,Z 435.825,A -85,B 0,C 180,E1 -23758.394,E2 -23758.394} C_VEL
LIN {X 0,Y 171.341,Z 434.461,A -85,B 0,C 180,E1 -23761.763,E2 -23761.763} C_VEL
LIN {X 0,Y 170.815,Z 433.935,A -85,B 0,C 180,E1 -23767.09,E2 -23767.09} C_VEL
LIN {X 0,Y 171.232,Z 434.951,A -85,B 0,C 180,E1 -23770.892,E2 -23770.892} C_VEL
LIN {X 0,Y 174.507,Z 437.687,A -85,B 0,C 180,E1 -23778.796,E2 -23778.796} C_VEL
LIN {X 0,Y 176.414,Z 441.152,A -85,B 0,C 180,E1 -23781.854,E2 -23781.854} C_VEL
LIN {X 0,Y 178.802,Z 443.197,A -85,B 0,C 180,E1 -23784.642,E2 -23784.642} C_VEL
LIN {X 0,Y 181.014,Z 446.6,A -85,B 0,C 180,E1 -23786.986,E2 -23786.986} C_VEL
LIN {X 0,Y 183.235,Z 449.557,A -85,B 0,C 180,E1 -23789.013,E2 -23789.013} C_VEL
LIN {X 0,Y 186.96,Z 455.331,A -85,B 0,C 180,E1 -23792.05,E2 -23792.05} C_VEL
LIN {X 0,Y 190.517,Z 461.116,A -85,B 0,C 180,E1 -23794.596,E2 -23794.596} C_VEL
LIN {X 0,Y 194.261,Z 467.729,A -85,B 0,C 180,E1 -23797.019,E2 -23797.019} C_VEL
LIN {X 0,Y 199.118,Z 477.164,A -85,B 0,C 180,E1 -23799.855,E2 -23799.855} C_VEL
LIN {X 0,Y 203.489,Z 486.748,A -85,B 0,C 180,E1 -23802.189,E2 -23802.189} C_VEL
LIN {X 0,Y 205.968,Z 492.868,A -85,B 0,C 180,E1 -23803.451,E2 -23803.451} C_VEL
LIN {X 0,Y 203.395,Z 526.573,A -85,B 0,C 180,E1 -23804.54,E2 -23804.54} C_VEL
LIN {X 0,Y 201.205,Z 540.305,A -85,B 0,C 180,E1 -23805.275,E2 -23805.275} C_VEL
LIN {X 0,Y 198.32,Z 552.719,A -85,B 0,C 180,E1 -23806.29,E2 -23806.29} C_VEL
LIN {X 0,Y 194.317,Z 565.152,A -85,B 0,C 180,E1 -23807.654,E2 -23807.654} C_VEL
LIN {X 0,Y 190.092,Z 576.226,A -85,B 0,C 180,E1 -23809.337,E2 -23809.337} C_VEL
LIN {X 0,Y 185.641,Z 586.212,A -85,B 0,C 180,E1 -23811.345,E2 -23811.345} C_VEL
LIN {X 0,Y 180.835,Z 595.262,A -85,B 0,C 180,E1 -23813.654,E2 -23813.654} C_VEL
LIN {X 0,Y 175.479,Z 604.101,A -85,B 0,C 180,E1 -23816.587,E2 -23816.587} C_VEL
LIN {X 0,Y 170.401,Z 611.767,A -85,B 0,C 180,E1 -23820.012,E2 -23820.012} C_VEL
LIN {X 0,Y 166.935,Z 616.571,A -85,B 0,C 180,E1 -23822.836,E2 -23822.836} C_VEL
LIN {X 0,Y 164.389,Z 619.106,A -85,B 0,C 180,E1 -23824.475,E2 -23824.475} C_VEL
LIN {X 0,Y 156.499,Z 623.874,A -85,B 0,C 180,E1 -23828.188,E2 -23828.188} C_VEL
LIN {X 0,Y 152.697,Z 625.953,A -85,B 0,C 180,E1 -23830.638,E2 -23830.638} C_VEL
LIN {X 0,Y 151.541,Z 626.783,A -85,B 0,C 180,E1 -23832.018,E2 -23832.018} C_VEL
LIN {X 0,Y 149.479,Z 628.69,A -85,B 0,C 180,E1 -23836.404,E2 -23836.404} C_VEL
LIN {X 0,Y 148.031,Z 629.547,A -85,B 0,C 180,E1 -23841.812,E2 -23841.812} C_VEL
LIN {X 0,Y 147.716,Z 629.364,A -85,B 0,C 180,E1 -23844.541,E2 -23844.541} C_VEL
LIN {X 0,Y 147.658,Z 627.832,A -85,B 0,C 180,E1 -23850.001,E2 -23850.001} C_VEL
LIN {X 0,Y 147.556,Z 626.467,A -85,B 0,C 180,E1 -23852.731,E2 -23852.731} C_VEL
LIN {X 0,Y 147.749,Z 623.563,A -85,B 0,C 180,E1 -23856.83,E2 -23856.83} C_VEL
LIN {X 0,Y 148.401,Z 619.606,A -85,B 0,C 180,E1 -23860.92,E2 -23860.92} C_VEL
LIN {X 0,Y 149.828,Z 613.487,A -85,B 0,C 180,E1 -23865.648,E2 -23865.648} C_VEL
LIN {X 0,Y 151.828,Z 606.775,A -85,B 0,C 180,E1 -23869.609,E2 -23869.609} C_VEL
LIN {X 0,Y 154.463,Z 598.426,A -85,B 0,C 180,E1 -23873.461,E2 -23873.461} C_VEL
LIN {X 0,Y 156.892,Z 589.798,A -85,B 0,C 180,E1 -23876.612,E2 -23876.612} C_VEL
LIN {X 0,Y 159.907,Z 579.134,A -85,B 0,C 180,E1 -23879.633,E2 -23879.633} C_VEL
LIN {X 0,Y 162.279,Z 569.992,A -85,B 0,C 180,E1 -23881.676,E2 -23881.676} C_VEL
LIN {X 0,Y 165.001,Z 558.718,A -85,B 0,C 180,E1 -23883.622,E2 -23883.622} C_VEL
LIN {X 0,Y 167.135,Z 547.239,A -85,B 0,C 180,E1 -23885.138,E2 -23885.138} C_VEL
LIN {X 0,Y 168.936,Z 534.277,A -85,B 0,C 180,E1 -23886.342,E2 -23886.342} C_VEL
LIN {X 0,Y 170.151,Z 521.388,A -85,B 0,C 180,E1 -23887.083,E2 -23887.083} C_VEL
LIN {X 0,Y 172.575,Z 473.203,A -85,B 0,C 180,E1 -23888.957,E2 -23888.957} C_VEL
LIN {X 0,Y 171.593,Z 465.469,A -85,B 0,C 180,E1 -23889.559,E2 -23889.559} C_VEL
LIN {X 0,Y 166.067,Z 450.286,A -85,B 0,C 180,E1 -23891.65,E2 -23891.65} C_VEL
LIN {X 0,Y 160.873,Z 438.581,A -85,B 0,C 180,E1 -23893.65,E2 -23893.65} C_VEL
LIN {X 0,Y 156.854,Z 431.465,A -85,B 0,C 180,E1 -23895.215,E2 -23895.215} C_VEL
LIN {X 0,Y 152.399,Z 424.466,A -85,B 0,C 180,E1 -23897.039,E2 -23897.039} C_VEL
LIN {X 0,Y 150.635,Z 421.796,A -85,B 0,C 180,E1 -23897.827,E2 -23897.827} C_VEL
LIN {X 0,Y 150.277,Z 420.565,A -85,B 0,C 180,E1 -23898.341,E2 -23898.341} C_VEL
LIN {X 0,Y 150.23,Z 420.268,A -85,B 0,C 180,E1 -23899.084,E2 -23899.084} C_VEL
LIN {X 0,Y 150.223,Z 420.258,A -85,B 0,C 180,E1 -23902.685,E2 -23902.685} C_VEL
LIN {X 0,Y 150.217,Z 420.277,A -85,B 0,C 180,E1 -23907.366,E2 -23907.366} C_VEL
LIN {X 0,Y 150.241,Z 420.249,A -85,B 0,C 180,E1 -23912.72,E2 -23912.72} C_VEL
LIN {X 0,Y 150.349,Z 420.221,A -85,B 0,C 180,E1 -23919.21,E2 -23919.21} C_VEL
LIN {X 0,Y 150.36,Z 420.253,A -85,B 0,C 180,E1 -23923.713,E2 -23923.713} C_VEL
LIN {X 0,Y 150.61,Z 420.181,A -85,B 0,C 180,E1 -23929.242,E2 -23929.242} C_VEL
LIN {X 0,Y 150.688,Z 420.185,A -85,B 0,C 180,E1 -23931.957,E2 -23931.957} C_VEL
LIN {X 0,Y 151.216,Z 420.102,A -85,B 0,C 180,E1 -23940,E2 -23940} C_VEL
LIN {X 0,Y 150.706,Z 420.207,A -85,B 0,C 180,E1 -23948.042,E2 -23948.042} C_VEL
LIN {X 0,Y 150.575,Z 420.182,A -85,B 0,C 180,E1 -23951.434,E2 -23951.434} C_VEL
LIN {X 0,Y 150.352,Z 420.243,A -85,B 0,C 180,E1 -23956.288,E2 -23956.288} C_VEL
LIN {X 0,Y 150.35,Z 420.235,A -85,B 0,C 180,E1 -23960.792,E2 -23960.792} C_VEL
LIN {X 0,Y 150.242,Z 420.259,A -85,B 0,C 180,E1 -23967.281,E2 -23967.281} C_VEL
LIN {X 0,Y 150.219,Z 420.237,A -85,B 0,C 180,E1 -23972.635,E2 -23972.635} C_VEL
LIN {X 0,Y 150.177,Z 420.276,A -85,B 0,C 180,E1 -23977.472,E2 -23977.472} C_VEL
LIN {X 0,Y 150.149,Z 420.253,A -85,B 0,C 180,E1 -23981.504,E2 -23981.504} C_VEL
LIN {X 0,Y 150.144,Z 420.282,A -85,B 0,C 180,E1 -23985.403,E2 -23985.403} C_VEL
LIN {X 0,Y 150.189,Z 420.256,A -85,B 0,C 180,E1 -23989.071,E2 -23989.071} C_VEL
LIN {X 0,Y 150.284,Z 420.36,A -85,B 0,C 180,E1 -23994.638,E2 -23994.638} C_VEL
LIN {X 0,Y 150.431,Z 421.181,A -85,B 0,C 180,E1 -23995.257,E2 -23995.257} C_VEL
LIN {X 0,Y 151.953,Z 424.007,A -85,B 0,C 180,E1 -23996.039,E2 -23996.039} C_VEL
LIN {X 0,Y 153.306,Z 425.857,A -85,B 0,C 180,E1 -23996.596,E2 -23996.596} C_VEL
LIN {X 0,Y 158.35,Z 433.814,A -85,B 0,C 180,E1 -23998.613,E2 -23998.613} C_VEL
LIN {X 0,Y 165.198,Z 445.802,A -85,B 0,C 180,E1 -24001.148,E2 -24001.148} C_VEL
LIN {X 0,Y 168.821,Z 454.271,A -85,B 0,C 180,E1 -24002.486,E2 -24002.486} C_VEL
LIN {X 0,Y 172.905,Z 465.827,A -85,B 0,C 180,E1 -24004.007,E2 -24004.007} C_VEL
LIN {X 0,Y 169.969,Z 520.817,A -85,B 0,C 180,E1 -24006.14,E2 -24006.14} C_VEL
LIN {X 0,Y 168.555,Z 533.857,A -85,B 0,C 180,E1 -24007.02,E2 -24007.02} C_VEL
LIN {X 0,Y 166.763,Z 545.516,A -85,B 0,C 180,E1 -24008.207,E2 -24008.207} C_VEL
LIN {X 0,Y 164.444,Z 558.079,A -85,B 0,C 180,E1 -24010.007,E2 -24010.007} C_VEL
LIN {X 0,Y 161.54,Z 569.91,A -85,B 0,C 180,E1 -24012.269,E2 -24012.269} C_VEL
LIN {X 0,Y 158.854,Z 579.429,A -85,B 0,C 180,E1 -24014.606,E2 -24014.606} C_VEL
LIN {X 0,Y 156.039,Z 589.133,A -85,B 0,C 180,E1 -24017.646,E2 -24017.646} C_VEL
LIN {X 0,Y 153.69,Z 597.078,A -85,B 0,C 180,E1 -24020.79,E2 -24020.79} C_VEL
LIN {X 0,Y 151.252,Z 604.864,A -85,B 0,C 180,E1 -24024.667,E2 -24024.667} C_VEL
LIN {X 0,Y 149.547,Z 611.089,A -85,B 0,C 180,E1 -24028.653,E2 -24028.653} C_VEL
LIN {X 0,Y 148.426,Z 616.036,A -85,B 0,C 180,E1 -24032.713,E2 -24032.713} C_VEL
LIN {X 0,Y 147.616,Z 619.868,A -85,B 0,C 180,E1 -24036.835,E2 -24036.835} C_VEL
LIN {X 0,Y 147.204,Z 622.666,A -85,B 0,C 180,E1 -24041.009,E2 -24041.009} C_VEL
LIN {X 0,Y 147.201,Z 623.985,A -85,B 0,C 180,E1 -24043.81,E2 -24043.81} C_VEL
LIN {X 0,Y 147.517,Z 625.106,A -85,B 0,C 180,E1 -24047.667,E2 -24047.667} C_VEL
LIN {X 0,Y 148.314,Z 625.42,A -85,B 0,C 180,E1 -24052.276,E2 -24052.276} C_VEL
LIN {X 0,Y 150.085,Z 624.516,A -85,B 0,C 180,E1 -24057.164,E2 -24057.164} C_VEL
LIN {X 0,Y 151.858,Z 623.052,A -85,B 0,C 180,E1 -24060.601,E2 -24060.601} C_VEL
LIN {X 0,Y 155.49,Z 619.577,A -85,B 0,C 180,E1 -24065.553,E2 -24065.553} C_VEL
LIN {X 0,Y 159.51,Z 615.122,A -85,B 0,C 180,E1 -24069.706,E2 -24069.706} C_VEL
LIN {X 0,Y 164.654,Z 608.672,A -85,B 0,C 180,E1 -24073.914,E2 -24073.914} C_VEL
LIN {X 0,Y 169.769,Z 601.602,A -85,B 0,C 180,E1 -24077.289,E2 -24077.289} C_VEL
LIN {X 0,Y 174.499,Z 594.334,A -85,B 0,C 180,E1 -24079.925,E2 -24079.925} C_VEL
LIN {X 0,Y 180.064,Z 584.448,A -85,B 0,C 180,E1 -24082.676,E2 -24082.676} C_VEL
LIN {X 0,Y 184.941,Z 574.447,A -85,B 0,C 180,E1 -24084.786,E2 -24084.786} C_VEL
LIN {X 0,Y 189.188,Z 563.998,A -85,B 0,C 180,E1 -24086.507,E2 -24086.507} C_VEL
LIN {X 0,Y 192.85,Z 552.873,A -85,B 0,C 180,E1 -24087.916,E2 -24087.916} C_VEL
LIN {X 0,Y 196.217,Z 540.334,A -85,B 0,C 180,E1 -24089.021,E2 -24089.021} C_VEL
LIN {X 0,Y 198.704,Z 527.057,A -85,B 0,C 180,E1 -24089.846,E2 -24089.846} C_VEL
LIN {X 0,Y 200.27,Z 512.225,A -85,B 0,C 180,E1 -24090.386,E2 -24090.386} C_VEL
LIN {X 0,Y 201.695,Z 492.178,A -85,B 0,C 180,E1 -24091.029,E2 -24091.029} C_VEL
LIN {X 0,Y 197.594,Z 482.821,A -85,B 0,C 180,E1 -24093.287,E2 -24093.287} C_VEL
LIN {X 0,Y 193.066,Z 473.85,A -85,B 0,C 180,E1 -24095.982,E2 -24095.982} C_VEL
LIN {X 0,Y 188.325,Z 465.477,A -85,B 0,C 180,E1 -24099.137,E2 -24099.137} C_VEL
LIN {X 0,Y 185.558,Z 461.501,A -85,B 0,C 180,E1 -24101.144,E2 -24101.144} C_VEL
LIN {X 0,Y 183.438,Z 458.452,A -85,B 0,C 180,E1 -24102.831,E2 -24102.831} C_VEL
LIN {X 0,Y 180.187,Z 453.917,A -85,B 0,C 180,E1 -24105.747,E2 -24105.747} C_VEL
LIN {X 0,Y 177.766,Z 450.775,A -85,B 0,C 180,E1 -24108.252,E2 -24108.252} C_VEL
LIN {X 0,Y 176.986,Z 449.428,A -85,B 0,C 180,E1 -24109.2,E2 -24109.2} C_VEL
LIN {X 0,Y 174.55,Z 446.687,A -85,B 0,C 180,E1 -24112.408,E2 -24112.408} C_VEL
LIN {X 0,Y 173.552,Z 444.465,A -85,B 0,C 180,E1 -24114.19,E2 -24114.19} C_VEL
LIN {X 0,Y 171.036,Z 442.392,A -85,B 0,C 180,E1 -24119.559,E2 -24119.559} C_VEL
LIN {X 0,Y 170.334,Z 441.372,A -85,B 0,C 180,E1 -24122.365,E2 -24122.365} C_VEL
LIN {X 0,Y 169.939,Z 440.994,A -85,B 0,C 180,E1 -24127.127,E2 -24127.127} C_VEL
LIN {X 0,Y 170.295,Z 441.948,A -85,B 0,C 180,E1 -24130.627,E2 -24130.627} C_VEL
LIN {X 0,Y 173.3,Z 444.665,A -85,B 0,C 180,E1 -24138.318,E2 -24138.318} C_VEL
LIN {X 0,Y 175.274,Z 448.158,A -85,B 0,C 180,E1 -24141.578,E2 -24141.578} C_VEL
LIN {X 0,Y 177.263,Z 449.94,A -85,B 0,C 180,E1 -24144.005,E2 -24144.005} C_VEL
LIN {X 0,Y 181.353,Z 456.038,A -85,B 0,C 180,E1 -24148.259,E2 -24148.259} C_VEL
LIN {X 0,Y 184.735,Z 461.455,A -85,B 0,C 180,E1 -24151.172,E2 -24151.172} C_VEL
LIN {X 0,Y 188.051,Z 467.089,A -85,B 0,C 180,E1 -24153.687,E2 -24153.687} C_VEL
LIN {X 0,Y 191.791,Z 473.99,A -85,B 0,C 180,E1 -24156.242,E2 -24156.242} C_VEL
LIN {X 0,Y 196.856,Z 484.349,A -85,B 0,C 180,E1 -24159.344,E2 -24159.344} C_VEL
LIN {X 0,Y 200.6,Z 493.24,A -85,B 0,C 180,E1 -24161.459,E2 -24161.459} C_VEL
LIN {X 0,Y 201.533,Z 495.987,A -85,B 0,C 180,E1 -24161.987,E2 -24161.987} C_VEL
LIN {X 0,Y 199.077,Z 526.057,A -85,B 0,C 180,E1 -24162.935,E2 -24162.935} C_VEL
LIN {X 0,Y 196.907,Z 539.489,A -85,B 0,C 180,E1 -24163.643,E2 -24163.643} C_VEL
LIN {X 0,Y 194.205,Z 551.127,A -85,B 0,C 180,E1 -24164.566,E2 -24164.566} C_VEL
LIN {X 0,Y 190.352,Z 563.152,A -85,B 0,C 180,E1 -24165.824,E2 -24165.824} C_VEL
LIN {X 0,Y 185.868,Z 574.586,A -85,B 0,C 180,E1 -24167.479,E2 -24167.479} C_VEL
LIN {X 0,Y 181.156,Z 584.887,A -85,B 0,C 180,E1 -24169.474,E2 -24169.474} C_VEL
LIN {X 0,Y 176.174,Z 594.188,A -85,B 0,C 180,E1 -24171.807,E2 -24171.807} C_VEL
LIN {X 0,Y 170.494,Z 603.192,A -85,B 0,C 180,E1 -24174.755,E2 -24174.755} C_VEL
LIN {X 0,Y 165.324,Z 610.678,A -85,B 0,C 180,E1 -24178.046,E2 -24178.046} C_VEL
LIN {X 0,Y 160.49,Z 617.009,A -85,B 0,C 180,E1 -24181.818,E2 -24181.818} C_VEL
LIN {X 0,Y 156.032,Z 622.209,A -85,B 0,C 180,E1 -24186.086,E2 -24186.086} C_VEL
LIN {X 0,Y 153.898,Z 624.472,A -85,B 0,C 180,E1 -24188.573,E2 -24188.573} C_VEL
LIN {X 0,Y 151.541,Z 626.783,A -85,B 0,C 180,E1 -24192.018,E2 -24192.018} C_VEL
LIN {X 0,Y 149.777,Z 627.904,A -85,B 0,C 180,E1 -24194.127,E2 -24194.127} C_VEL
LIN {X 0,Y 145.505,Z 629.056,A -85,B 0,C 180,E1 -24197.572,E2 -24197.572} C_VEL
LIN {X 0,Y 142.294,Z 629.416,A -85,B 0,C 180,E1 -24200.471,E2 -24200.471} C_VEL
LIN {X 0,Y 140.866,Z 629.373,A -85,B 0,C 180,E1 -24202.8,E2 -24202.8} C_VEL
LIN {X 0,Y 140.697,Z 629.269,A -85,B 0,C 180,E1 -24203.601,E2 -24203.601} C_VEL
LIN {X 0,Y 140.491,Z 628.613,A -85,B 0,C 180,E1 -24207.133,E2 -24207.133} C_VEL
LIN {X 0,Y 140.561,Z 627.624,A -85,B 0,C 180,E1 -24210.001,E2 -24210.001} C_VEL
LIN {X 0,Y 140.481,Z 626.211,A -85,B 0,C 180,E1 -24212.868,E2 -24212.868} C_VEL
LIN {X 0,Y 140.676,Z 623.249,A -85,B 0,C 180,E1 -24217.175,E2 -24217.175} C_VEL
LIN {X 0,Y 141.408,Z 619.223,A -85,B 0,C 180,E1 -24221.467,E2 -24221.467} C_VEL
LIN {X 0,Y 142.947,Z 612.994,A -85,B 0,C 180,E1 -24226.422,E2 -24226.422} C_VEL
LIN {X 0,Y 145.122,Z 606.196,A -85,B 0,C 180,E1 -24230.555,E2 -24230.555} C_VEL
LIN {X 0,Y 147.399,Z 599.247,A -85,B 0,C 180,E1 -24233.909,E2 -24233.909} C_VEL
LIN {X 0,Y 150.025,Z 590.591,A -85,B 0,C 180,E1 -24237.281,E2 -24237.281} C_VEL
LIN {X 0,Y 153.076,Z 580.499,A -85,B 0,C 180,E1 -24240.333,E2 -24240.333} C_VEL
LIN {X 0,Y 155.848,Z 570.221,A -85,B 0,C 180,E1 -24242.761,E2 -24242.761} C_VEL
LIN {X 0,Y 158.698,Z 559.029,A -85,B 0,C 180,E1 -24244.762,E2 -24244.762} C_VEL
LIN {X 0,Y 160.923,Z 547.665,A -85,B 0,C 180,E1 -24246.321,E2 -24246.321} C_VEL
LIN {X 0,Y 162.787,Z 535.131,A -85,B 0,C 180,E1 -24247.548,E2 -24247.548} C_VEL
LIN {X 0,Y 164.083,Z 521.975,A -85,B 0,C 180,E1 -24248.353,E2 -24248.353} C_VEL
LIN {X 0,Y 166.662,Z 474.021,A -85,B 0,C 180,E1 -24250.262,E2 -24250.262} C_VEL
LIN {X 0,Y 165.882,Z 467.835,A -85,B 0,C 180,E1 -24250.771,E2 -24250.771} C_VEL
LIN {X 0,Y 160.524,Z 452.942,A -85,B 0,C 180,E1 -24252.948,E2 -24252.948} C_VEL
LIN {X 0,Y 155.566,Z 441.736,A -85,B 0,C 180,E1 -24255.005,E2 -24255.005} C_VEL
LIN {X 0,Y 150.631,Z 433.181,A -85,B 0,C 180,E1 -24257.085,E2 -24257.085} C_VEL
LIN {X 0,Y 147.66,Z 428.782,A -85,B 0,C 180,E1 -24258.391,E2 -24258.391} C_VEL
LIN {X 0,Y 145.801,Z 425.829,A -85,B 0,C 180,E1 -24259.263,E2 -24259.263} C_VEL
LIN {X 0,Y 143.908,Z 423.612,A -85,B 0,C 180,E1 -24260.135,E2 -24260.135} C_VEL
LIN {X 0,Y 143.217,Z 421.62,A -85,B 0,C 180,E1 -24260.783,E2 -24260.783} C_VEL
LIN {X 0,Y 143.157,Z 421.164,A -85,B 0,C 180,E1 -24261.765,E2 -24261.765} C_VEL
LIN {X 0,Y 143.185,Z 421.153,A -85,B 0,C 180,E1 -24267.322,E2 -24267.322} C_VEL
LIN {X 0,Y 143.188,Z 421.122,A -85,B 0,C 180,E1 -24272.065,E2 -24272.065} C_VEL
LIN {X 0,Y 143.274,Z 421.103,A -85,B 0,C 180,E1 -24278.748,E2 -24278.748} C_VEL
LIN {X 0,Y 143.294,Z 421.124,A -85,B 0,C 180,E1 -24282.886,E2 -24282.886} C_VEL
LIN {X 0,Y 143.536,Z 421.062,A -85,B 0,C 180,E1 -24288.705,E2 -24288.705} C_VEL
LIN {X 0,Y 143.612,Z 421.059,A -85,B 0,C 180,E1 -24291.558,E2 -24291.558} C_VEL
LIN {X 0,Y 144.175,Z 420.977,A -85,B 0,C 180,E1 -24300,E2 -24300} C_VEL
LIN {X 0,Y 143.626,Z 421.083,A -85,B 0,C 180,E1 -24308.441,E2 -24308.441} C_VEL
LIN {X 0,Y 143.501,Z 421.06,A -85,B 0,C 180,E1 -24311.623,E2 -24311.623} C_VEL
LIN {X 0,Y 143.295,Z 421.131,A -85,B 0,C 180,E1 -24317.114,E2 -24317.114} C_VEL
LIN {X 0,Y 143.276,Z 421.106,A -85,B 0,C 180,E1 -24321.254,E2 -24321.254} C_VEL
LIN {X 0,Y 143.19,Z 421.143,A -85,B 0,C 180,E1 -24327.937,E2 -24327.937} C_VEL
LIN {X 0,Y 143.146,Z 421.115,A -85,B 0,C 180,E1 -24333.422,E2 -24333.422} C_VEL
LIN {X 0,Y 143.062,Z 421.149,A -85,B 0,C 180,E1 -24339.69,E2 -24339.69} C_VEL
LIN {X 0,Y 143.062,Z 421.14,A -85,B 0,C 180,E1 -24343.453,E2 -24343.453} C_VEL
LIN {X 0,Y 143.089,Z 421.147,A -85,B 0,C 180,E1 -24347.455,E2 -24347.455} C_VEL
LIN {X 0,Y 143.223,Z 421.394,A -85,B 0,C 180,E1 -24352.318,E2 -24352.318} C_VEL
LIN {X 0,Y 143.546,Z 422.634,A -85,B 0,C 180,E1 -24352.889,E2 -24352.889} C_VEL
LIN {X 0,Y 145.107,Z 425.165,A -85,B 0,C 180,E1 -24353.686,E2 -24353.686} C_VEL
LIN {X 0,Y 146.313,Z 426.538,A -85,B 0,C 180,E1 -24354.227,E2 -24354.227} C_VEL
LIN {X 0,Y 148.597,Z 429.967,A -85,B 0,C 180,E1 -24355.269,E2 -24355.269} C_VEL
LIN {X 0,Y 155.309,Z 440.849,A -85,B 0,C 180,E1 -24358.119,E2 -24358.119} C_VEL
LIN {X 0,Y 161.453,Z 452.383,A -85,B 0,C 180,E1 -24360.527,E2 -24360.527} C_VEL
LIN {X 0,Y 166.718,Z 466.664,A -85,B 0,C 180,E1 -24362.625,E2 -24362.625} C_VEL
LIN {X 0,Y 166.94,Z 469.364,A -85,B 0,C 180,E1 -24362.819,E2 -24362.819} C_VEL
LIN {X 0,Y 163.902,Z 521.415,A -85,B 0,C 180,E1 -24364.873,E2 -24364.873} C_VEL
LIN {X 0,Y 162.398,Z 534.654,A -85,B 0,C 180,E1 -24365.814,E2 -24365.814} C_VEL
LIN {X 0,Y 160.441,Z 546.607,A -85,B 0,C 180,E1 -24367.09,E2 -24367.09} C_VEL
LIN {X 0,Y 158.189,Z 558.196,A -85,B 0,C 180,E1 -24368.822,E2 -24368.822} C_VEL
LIN {X 0,Y 155.142,Z 570.089,A -85,B 0,C 180,E1 -24371.169,E2 -24371.169} C_VEL
LIN {X 0,Y 152.332,Z 579.596,A -85,B 0,C 180,E1 -24373.585,E2 -24373.585} C_VEL
LIN {X 0,Y 149.69,Z 588.391,A -85,B 0,C 180,E1 -24376.423,E2 -24376.423} C_VEL
LIN {X 0,Y 147.127,Z 596.481,A -85,B 0,C 180,E1 -24379.68,E2 -24379.68} C_VEL
LIN {X 0,Y 144.521,Z 604.432,A -85,B 0,C 180,E1 -24383.718,E2 -24383.718} C_VEL
LIN {X 0,Y 142.972,Z 609.799,A -85,B 0,C 180,E1 -24387.182,E2 -24387.182} C_VEL
LIN {X 0,Y 141.614,Z 615.058,A -85,B 0,C 180,E1 -24391.421,E2 -24391.421} C_VEL
LIN {X 0,Y 140.709,Z 619.153,A -85,B 0,C 180,E1 -24395.732,E2 -24395.732} C_VEL
LIN {X 0,Y 140.254,Z 621.281,A -85,B 0,C 180,E1 -24398.645,E2 -24398.645} C_VEL
LIN {X 0,Y 140.075,Z 622.967,A -85,B 0,C 180,E1 -24401.576,E2 -24401.576} C_VEL
LIN {X 0,Y 140.143,Z 624.242,A -85,B 0,C 180,E1 -24404.52,E2 -24404.52} C_VEL
LIN {X 0,Y 140.466,Z 625.19,A -85,B 0,C 180,E1 -24408.079,E2 -24408.079} C_VEL
LIN {X 0,Y 141.484,Z 625.502,A -85,B 0,C 180,E1 -24413.414,E2 -24413.414} C_VEL
LIN {X 0,Y 143.248,Z 624.662,A -85,B 0,C 180,E1 -24417.98,E2 -24417.98} C_VEL
LIN {X 0,Y 145.513,Z 622.957,A -85,B 0,C 180,E1 -24422.09,E2 -24422.09} C_VEL
LIN {X 0,Y 149.079,Z 619.779,A -85,B 0,C 180,E1 -24426.733,E2 -24426.733} C_VEL
LIN {X 0,Y 152.437,Z 616.327,A -85,B 0,C 180,E1 -24430.198,E2 -24430.198} C_VEL
LIN {X 0,Y 157.575,Z 610.476,A -85,B 0,C 180,E1 -24434.47,E2 -24434.47} C_VEL
LIN {X 0,Y 162.958,Z 603.579,A -85,B 0,C 180,E1 -24438.067,E2 -24438.067} C_VEL
LIN {X 0,Y 168.993,Z 594.895,A -85,B 0,C 180,E1 -24441.405,E2 -24441.405} C_VEL
LIN {X 0,Y 174.591,Z 585.508,A -85,B 0,C 180,E1 -24444.104,E2 -24444.104} C_VEL
LIN {X 0,Y 180.02,Z 574.914,A -85,B 0,C 180,E1 -24446.383,E2 -24446.383} C_VEL
LIN {X 0,Y 184.87,Z 563.408,A -85,B 0,C 180,E1 -24448.275,E2 -24448.275} C_VEL
LIN {X 0,Y 188.766,Z 551.869,A -85,B 0,C 180,E1 -24449.686,E2 -24449.686} C_VEL
LIN {X 0,Y 192.229,Z 538.981,A -85,B 0,C 180,E1 -24450.792,E2 -24450.792} C_VEL
LIN {X 0,Y 194.62,Z 526,A -85,B 0,C 180,E1 -24451.558,E2 -24451.558} C_VEL
LIN {X 0,Y 196.229,Z 510.341,A -85,B 0,C 180,E1 -24452.107,E2 -24452.107} C_VEL
LIN {X 0,Y 197.384,Z 495.032,A -85,B 0,C 180,E1 -24452.594,E2 -24452.594} C_VEL
LIN {X 0,Y 193.444,Z 485.861,A -85,B 0,C 180,E1 -24454.954,E2 -24454.954} C_VEL
LIN {X 0,Y 188.536,Z 476.128,A -85,B 0,C 180,E1 -24458.169,E2 -24458.169} C_VEL
LIN {X 0,Y 185.612,Z 471.018,A -85,B 0,C 180,E1 -24460.284,E2 -24460.284} C_VEL
LIN {X 0,Y 181.637,Z 464.984,A -85,B 0,C 180,E1 -24463.481,E2 -24463.481} C_VEL
LIN {X 0,Y 178.419,Z 460.435,A -85,B 0,C 180,E1 -24466.507,E2 -24466.507} C_VEL
LIN {X 0,Y 175.737,Z 456.464,A -85,B 0,C 180,E1 -24469.546,E2 -24469.546} C_VEL
LIN {X 0,Y 172.985,Z 452.947,A -85,B 0,C 180,E1 -24473.439,E2 -24473.439} C_VEL
LIN {X 0,Y 172.317,Z 451.37,A -85,B 0,C 180,E1 -24474.735,E2 -24474.735} C_VEL
LIN {X 0,Y 169.933,Z 449.129,A -85,B 0,C 180,E1 -24480.296,E2 -24480.296} C_VEL
LIN {X 0,Y 169.451,Z 448.434,A -85,B 0,C 180,E1 -24482.377,E2 -24482.377} C_VEL
LIN {X 0,Y 169.096,Z 448.167,A -85,B 0,C 180,E1 -24487.886,E2 -24487.886} C_VEL
LIN {X 0,Y 172.131,Z 451.615,A -85,B 0,C 180,E1 -24497.87,E2 -24497.87} C_VEL
LIN {X 0,Y 174.015,Z 455.006,A -85,B 0,C 180,E1 -24501.124,E2 -24501.124} C_VEL
LIN {X 0,Y 175.824,Z 456.799,A -85,B 0,C 180,E1 -24503.446,E2 -24503.446} C_VEL
LIN {X 0,Y 179.425,Z 462.33,A -85,B 0,C 180,E1 -24507.399,E2 -24507.399} C_VEL
LIN {X 0,Y 182.638,Z 467.752,A -85,B 0,C 180,E1 -24510.348,E2 -24510.348} C_VEL
LIN {X 0,Y 185.985,Z 473.653,A -85,B 0,C 180,E1 -24513.017,E2 -24513.017} C_VEL
LIN {X 0,Y 190.454,Z 482.477,A -85,B 0,C 180,E1 -24516.187,E2 -24516.187} C_VEL
LIN {X 0,Y 194.945,Z 492.455,A -85,B 0,C 180,E1 -24519.033,E2 -24519.033} C_VEL
LIN {X 0,Y 197.194,Z 498.268,A -85,B 0,C 180,E1 -24520.385,E2 -24520.385} C_VEL
LIN {X 0,Y 194.801,Z 526.426,A -85,B 0,C 180,E1 -24521.297,E2 -24521.297} C_VEL
LIN {X 0,Y 192.418,Z 540.305,A -85,B 0,C 180,E1 -24522.032,E2 -24522.032} C_VEL
LIN {X 0,Y 189.642,Z 551.671,A -85,B 0,C 180,E1 -24522.954,E2 -24522.954} C_VEL
LIN {X 0,Y 185.952,Z 562.729,A -85,B 0,C 180,E1 -24524.104,E2 -24524.104} C_VEL
LIN {X 0,Y 181.327,Z 574.219,A -85,B 0,C 180,E1 -24525.763,E2 -24525.763} C_VEL
LIN {X 0,Y 176.342,Z 584.577,A -85,B 0,C 180,E1 -24527.738,E2 -24527.738} C_VEL
LIN {X 0,Y 171.735,Z 593.044,A -85,B 0,C 180,E1 -24529.87,E2 -24529.87} C_VEL
LIN {X 0,Y 166.696,Z 600.893,A -85,B 0,C 180,E1 -24532.316,E2 -24532.316} C_VEL
LIN {X 0,Y 161.164,Z 608.585,A -85,B 0,C 180,E1 -24535.467,E2 -24535.467} C_VEL
LIN {X 0,Y 155.866,Z 615.418,A -85,B 0,C 180,E1 -24539.322,E2 -24539.322} C_VEL
LIN {X 0,Y 150.819,Z 621.104,A -85,B 0,C 180,E1 -24543.726,E2 -24543.726} C_VEL
LIN {X 0,Y 147.317,Z 624.583,A -85,B 0,C 180,E1 -24547.565,E2 -24547.565} C_VEL
LIN {X 0,Y 144.626,Z 626.953,A -85,B 0,C 180,E1 -24551.425,E2 -24551.425} C_VEL
LIN {X 0,Y 142.584,Z 628.667,A -85,B 0,C 180,E1 -24555.733,E2 -24555.733} C_VEL
LIN {X 0,Y 141.646,Z 629.254,A -85,B 0,C 180,E1 -24558.554,E2 -24558.554} C_VEL
LIN {X 0,Y 140.697,Z 629.269,A -85,B 0,C 180,E1 -24563.601,E2 -24563.601} C_VEL
LIN {X 0,Y 140.253,Z 629.064,A -85,B 0,C 180,E1 -24565.194,E2 -24565.194} C_VEL
LIN {X 0,Y 138.791,Z 628.483,A -85,B 0,C 180,E1 -24567.543,E2 -24567.543} C_VEL
LIN {X 0,Y 135.588,Z 626.852,A -85,B 0,C 180,E1 -24571.438,E2 -24571.438} C_VEL
LIN {X 0,Y 133.743,Z 624.968,A -85,B 0,C 180,E1 -24574.665,E2 -24574.665} C_VEL
LIN {X 0,Y 133.521,Z 623.825,A -85,B 0,C 180,E1 -24576.308,E2 -24576.308} C_VEL
LIN {X 0,Y 134.094,Z 620.285,A -85,B 0,C 180,E1 -24580.571,E2 -24580.571} C_VEL
LIN {X 0,Y 135.307,Z 615.409,A -85,B 0,C 180,E1 -24585.053,E2 -24585.053} C_VEL
LIN {X 0,Y 137.196,Z 609.239,A -85,B 0,C 180,E1 -24589.449,E2 -24589.449} C_VEL
LIN {X 0,Y 139.797,Z 601.544,A -85,B 0,C 180,E1 -24593.715,E2 -24593.715} C_VEL
LIN {X 0,Y 141.974,Z 595.327,A -85,B 0,C 180,E1 -24596.457,E2 -24596.457} C_VEL
LIN {X 0,Y 144.913,Z 586.085,A -85,B 0,C 180,E1 -24599.809,E2 -24599.809} C_VEL
LIN {X 0,Y 147.981,Z 575.799,A -85,B 0,C 180,E1 -24602.699,E2 -24602.699} C_VEL
LIN {X 0,Y 151.152,Z 564.387,A -85,B 0,C 180,E1 -24605.127,E2 -24605.127} C_VEL
LIN {X 0,Y 153.867,Z 552.511,A -85,B 0,C 180,E1 -24607.038,E2 -24607.038} C_VEL
LIN {X 0,Y 156.031,Z 540.167,A -85,B 0,C 180,E1 -24608.473,E2 -24608.473} C_VEL
LIN {X 0,Y 157.806,Z 526.258,A -85,B 0,C 180,E1 -24609.517,E2 -24609.517} C_VEL
LIN {X 0,Y 160.835,Z 474.811,A -85,B 0,C 180,E1 -24611.659,E2 -24611.659} C_VEL
LIN {X 0,Y 160.157,Z 469.849,A -85,B 0,C 180,E1 -24612.108,E2 -24612.108} C_VEL
LIN {X 0,Y 154.847,Z 455.103,A -85,B 0,C 180,E1 -24614.432,E2 -24614.432} C_VEL
LIN {X 0,Y 150.293,Z 444.767,A -85,B 0,C 180,E1 -24616.477,E2 -24616.477} C_VEL
LIN {X 0,Y 145.399,Z 436.513,A -85,B 0,C 180,E1 -24618.698,E2 -24618.698} C_VEL
LIN {X 0,Y 141.674,Z 430.958,A -85,B 0,C 180,E1 -24620.5,E2 -24620.5} C_VEL
LIN {X 0,Y 139.352,Z 427.504,A -85,B 0,C 180,E1 -24621.7,E2 -24621.7} C_VEL
LIN {X 0,Y 136.738,Z 424.283,A -85,B 0,C 180,E1 -24623.079,E2 -24623.079} C_VEL
LIN {X 0,Y 136.21,Z 422.738,A -85,B 0,C 180,E1 -24623.603,E2 -24623.603} C_VEL
LIN {X 0,Y 136.067,Z 422.076,A -85,B 0,C 180,E1 -24624.473,E2 -24624.473} C_VEL
LIN {X 0,Y 136.063,Z 422.022,A -85,B 0,C 180,E1 -24628.9,E2 -24628.9} C_VEL
LIN {X 0,Y 136.144,Z 422,A -85,B 0,C 180,E1 -24632.315,E2 -24632.315} C_VEL
LIN {X 0,Y 136.241,Z 421.977,A -85,B 0,C 180,E1 -24638.832,E2 -24638.832} C_VEL
LIN {X 0,Y 136.266,Z 422.01,A -85,B 0,C 180,E1 -24645.055,E2 -24645.055} C_VEL
LIN {X 0,Y 136.43,Z 421.949,A -85,B 0,C 180,E1 -24648.166,E2 -24648.166} C_VEL
LIN {X 0,Y 136.541,Z 421.935,A -85,B 0,C 180,E1 -24651.117,E2 -24651.117} C_VEL
LIN {X 0,Y 137.132,Z 421.853,A -85,B 0,C 180,E1 -24660,E2 -24660} C_VEL
LIN {X 0,Y 136.551,Z 421.955,A -85,B 0,C 180,E1 -24668.882,E2 -24668.882} C_VEL
LIN {X 0,Y 136.417,Z 421.94,A -85,B 0,C 180,E1 -24671.892,E2 -24671.892} C_VEL
LIN {X 0,Y 136.238,Z 422.014,A -85,B 0,C 180,E1 -24678.03,E2 -24678.03} C_VEL
LIN {X 0,Y 136.197,Z 421.98,A -85,B 0,C 180,E1 -24681.748,E2 -24681.748} C_VEL
LIN {X 0,Y 136.117,Z 422.028,A -85,B 0,C 180,E1 -24688.629,E2 -24688.629} C_VEL
LIN {X 0,Y 136.044,Z 422.001,A -85,B 0,C 180,E1 -24694.629,E2 -24694.629} C_VEL
LIN {X 0,Y 136.033,Z 422.03,A -85,B 0,C 180,E1 -24699.199,E2 -24699.199} C_VEL
LIN {X 0,Y 136.003,Z 422.019,A -85,B 0,C 180,E1 -24703.66,E2 -24703.66} C_VEL
LIN {X 0,Y 136.053,Z 422.196,A -85,B 0,C 180,E1 -24709.147,E2 -24709.147} C_VEL
LIN {X 0,Y 136.295,Z 423.172,A -85,B 0,C 180,E1 -24709.84,E2 -24709.84} C_VEL
LIN {X 0,Y 137.86,Z 425.938,A -85,B 0,C 180,E1 -24710.8,E2 -24710.8} C_VEL
LIN {X 0,Y 139.437,Z 427.54,A -85,B 0,C 180,E1 -24711.594,E2 -24711.594} C_VEL
LIN {X 0,Y 141.7,Z 430.952,A -85,B 0,C 180,E1 -24712.765,E2 -24712.765} C_VEL
LIN {X 0,Y 145.496,Z 436.807,A -85,B 0,C 180,E1 -24714.613,E2 -24714.613} C_VEL
LIN {X 0,Y 149.732,Z 443.618,A -85,B 0,C 180,E1 -24716.523,E2 -24716.523} C_VEL
LIN {X 0,Y 156.284,Z 455.756,A -85,B 0,C 180,E1 -24719.282,E2 -24719.282} C_VEL
LIN {X 0,Y 161.111,Z 469.232,A -85,B 0,C 180,E1 -24721.363,E2 -24721.363} C_VEL
LIN {X 0,Y 157.942,Z 521.835,A -85,B 0,C 180,E1 -24723.51,E2 -24723.51} C_VEL
LIN {X 0,Y 156.285,Z 535.594,A -85,B 0,C 180,E1 -24724.531,E2 -24724.531} C_VEL
LIN {X 0,Y 154.129,Z 548.152,A -85,B 0,C 180,E1 -24725.954,E2 -24725.954} C_VEL
LIN {X 0,Y 151.577,Z 559.911,A -85,B 0,C 180,E1 -24727.833,E2 -24727.833} C_VEL
LIN {X 0,Y 148.381,Z 571.548,A -85,B 0,C 180,E1 -24730.277,E2 -24730.277} C_VEL
LIN {X 0,Y 145.863,Z 579.739,A -85,B 0,C 180,E1 -24732.474,E2 -24732.474} C_VEL
LIN {X 0,Y 142.757,Z 589.427,A -85,B 0,C 180,E1 -24735.75,E2 -24735.75} C_VEL
LIN {X 0,Y 140.139,Z 597.359,A -85,B 0,C 180,E1 -24739.16,E2 -24739.16} C_VEL
LIN {X 0,Y 137.44,Z 605.125,A -85,B 0,C 180,E1 -24743.393,E2 -24743.393} C_VEL
LIN {X 0,Y 135.853,Z 610.419,A -85,B 0,C 180,E1 -24747.034,E2 -24747.034} C_VEL
LIN {X 0,Y 134.463,Z 615.557,A -85,B 0,C 180,E1 -24751.497,E2 -24751.497} C_VEL
LIN {X 0,Y 133.537,Z 619.556,A -85,B 0,C 180,E1 -24756.041,E2 -24756.041} C_VEL
LIN {X 0,Y 133.121,Z 621.621,A -85,B 0,C 180,E1 -24759.112,E2 -24759.112} C_VEL
LIN {X 0,Y 132.959,Z 623.263,A -85,B 0,C 180,E1 -24762.205,E2 -24762.205} C_VEL
LIN {X 0,Y 133.072,Z 624.489,A -85,B 0,C 180,E1 -24765.31,E2 -24765.31} C_VEL
LIN {X 0,Y 133.403,Z 625.269,A -85,B 0,C 180,E1 -24768.508,E2 -24768.508} C_VEL
LIN {X 0,Y 134.72,Z 625.585,A -85,B 0,C 180,E1 -24774.665,E2 -24774.665} C_VEL
LIN {X 0,Y 136.482,Z 624.8,A -85,B 0,C 180,E1 -24778.908,E2 -24778.908} C_VEL
LIN {X 0,Y 139.266,Z 622.863,A -85,B 0,C 180,E1 -24783.717,E2 -24783.717} C_VEL
LIN {X 0,Y 142.751,Z 619.973,A -85,B 0,C 180,E1 -24788.027,E2 -24788.027} C_VEL
LIN {X 0,Y 146.839,Z 616.042,A -85,B 0,C 180,E1 -24792.07,E2 -24792.07} C_VEL
LIN {X 0,Y 151.812,Z 610.702,A -85,B 0,C 180,E1 -24796.02,E2 -24796.02} C_VEL
LIN {X 0,Y 157.133,Z 604.284,A -85,B 0,C 180,E1 -24799.493,E2 -24799.493} C_VEL
LIN {X 0,Y 162.481,Z 597.114,A -85,B 0,C 180,E1 -24802.404,E2 -24802.404} C_VEL
LIN {X 0,Y 168.697,Z 587.494,A -85,B 0,C 180,E1 -24805.363,E2 -24805.363} C_VEL
LIN {X 0,Y 173.873,Z 578.161,A -85,B 0,C 180,E1 -24807.538,E2 -24807.538} C_VEL
LIN {X 0,Y 178.669,Z 567.95,A -85,B 0,C 180,E1 -24809.359,E2 -24809.359} C_VEL
LIN {X 0,Y 182.954,Z 556.692,A -85,B 0,C 180,E1 -24810.914,E2 -24810.914} C_VEL
LIN {X 0,Y 186.82,Z 544.253,A -85,B 0,C 180,E1 -24812.131,E2 -24812.131} C_VEL
LIN {X 0,Y 189.702,Z 531.355,A -85,B 0,C 180,E1 -24813.019,E2 -24813.019} C_VEL
LIN {X 0,Y 191.526,Z 518.804,A -85,B 0,C 180,E1 -24813.558,E2 -24813.558} C_VEL
LIN {X 0,Y 193.275,Z 498.018,A -85,B 0,C 180,E1 -24814.201,E2 -24814.201} C_VEL
LIN {X 0,Y 189.51,Z 489.204,A -85,B 0,C 180,E1 -24816.65,E2 -24816.65} C_VEL
LIN {X 0,Y 185.398,Z 480.901,A -85,B 0,C 180,E1 -24819.577,E2 -24819.577} C_VEL
LIN {X 0,Y 182.684,Z 475.95,A -85,B 0,C 180,E1 -24821.713,E2 -24821.713} C_VEL
LIN {X 0,Y 179.419,Z 471.033,A -85,B 0,C 180,E1 -24824.536,E2 -24824.536} C_VEL
LIN {X 0,Y 176.703,Z 466.916,A -85,B 0,C 180,E1 -24827.269,E2 -24827.269} C_VEL
LIN {X 0,Y 173.883,Z 462.722,A -85,B 0,C 180,E1 -24830.696,E2 -24830.696} C_VEL
LIN {X 0,Y 171.513,Z 459.29,A -85,B 0,C 180,E1 -24834.415,E2 -24834.415} C_VEL
LIN {X 0,Y 171.099,Z 458.262,A -85,B 0,C 180,E1 -24835.288,E2 -24835.288} C_VEL
LIN {X 0,Y 168.569,Z 455.49,A -85,B 0,C 180,E1 -24842.39,E2 -24842.39} C_VEL
LIN {X 0,Y 168.221,Z 455.233,A -85,B 0,C 180,E1 -24847.927,E2 -24847.927} C_VEL
LIN {X 0,Y 170.941,Z 458.558,A -85,B 0,C 180,E1 -24857.361,E2 -24857.361} C_VEL
LIN {X 0,Y 173.038,Z 462.167,A -85,B 0,C 180,E1 -24861.057,E2 -24861.057} C_VEL
LIN {X 0,Y 174.372,Z 463.518,A -85,B 0,C 180,E1 -24862.826,E2 -24862.826} C_VEL
LIN {X 0,Y 177.562,Z 468.655,A -85,B 0,C 180,E1 -24866.545,E2 -24866.545} C_VEL
LIN {X 0,Y 180.534,Z 473.926,A -85,B 0,C 180,E1 -24869.449,E2 -24869.449} C_VEL
LIN {X 0,Y 183.449,Z 479.287,A -85,B 0,C 180,E1 -24871.936,E2 -24871.936} C_VEL
LIN {X 0,Y 187.082,Z 486.825,A -85,B 0,C 180,E1 -24874.722,E2 -24874.722} C_VEL
LIN {X 0,Y 190.955,Z 495.63,A -85,B 0,C 180,E1 -24877.393,E2 -24877.393} C_VEL
LIN {X 0,Y 192.953,Z 500.716,A -85,B 0,C 180,E1 -24878.687,E2 -24878.687} C_VEL
LIN {X 0,Y 190.725,Z 526.677,A -85,B 0,C 180,E1 -24879.579,E2 -24879.579} C_VEL
LIN {X 0,Y 188.316,Z 540.242,A -85,B 0,C 180,E1 -24880.298,E2 -24880.298} C_VEL
LIN {X 0,Y 185.234,Z 552.213,A -85,B 0,C 180,E1 -24881.263,E2 -24881.263} C_VEL
LIN {X 0,Y 181.111,Z 563.905,A -85,B 0,C 180,E1 -24882.501,E2 -24882.501} C_VEL
LIN {X 0,Y 176.354,Z 575.153,A -85,B 0,C 180,E1 -24884.168,E2 -24884.168} C_VEL
LIN {X 0,Y 171.189,Z 585.325,A -85,B 0,C 180,E1 -24886.151,E2 -24886.151} C_VEL
LIN {X 0,Y 165.296,Z 595.278,A -85,B 0,C 180,E1 -24888.776,E2 -24888.776} C_VEL
LIN {X 0,Y 159.138,Z 604.064,A -85,B 0,C 180,E1 -24891.811,E2 -24891.811} C_VEL
LIN {X 0,Y 153.633,Z 611.132,A -85,B 0,C 180,E1 -24895.125,E2 -24895.125} C_VEL
LIN {X 0,Y 148.817,Z 616.785,A -85,B 0,C 180,E1 -24898.704,E2 -24898.704} C_VEL
LIN {X 0,Y 144.474,Z 621.263,A -85,B 0,C 180,E1 -24902.477,E2 -24902.477} C_VEL
LIN {X 0,Y 140.759,Z 624.684,A -85,B 0,C 180,E1 -24906.458,E2 -24906.458} C_VEL
LIN {X 0,Y 138.661,Z 626.398,A -85,B 0,C 180,E1 -24909.22,E2 -24909.22} C_VEL
LIN {X 0,Y 135.683,Z 628.646,A -85,B 0,C 180,E1 -24914.991,E2 -24914.991} C_VEL
LIN {X 0,Y 134.666,Z 629.196,A -85,B 0,C 180,E1 -24917.952,E2 -24917.952} C_VEL
LIN {X 0,Y 133.57,Z 629.069,A -85,B 0,C 180,E1 -24923.96,E2 -24923.96} C_VEL
LIN {X 0,Y 133.403,Z 628.433,A -85,B 0,C 180,E1 -24926.981,E2 -24926.981} C_VEL
LIN {X 0,Y 133.475,Z 627.413,A -85,B 0,C 180,E1 -24930.001,E2 -24930.001} C_VEL
LIN {X 0,Y 133.395,Z 625.936,A -85,B 0,C 180,E1 -24933.021,E2 -24933.021} C_VEL
LIN {X 0,Y 133.521,Z 623.825,A -85,B 0,C 180,E1 -24936.308,E2 -24936.308} C_VEL
LIN {X 0,Y 133.083,Z 621.978,A -85,B 0,C 180,E1 -24938.707,E2 -24938.707} C_VEL
LIN {X 0,Y 130.955,Z 618.373,A -85,B 0,C 180,E1 -24942.614,E2 -24942.614} C_VEL
LIN {X 0,Y 129.29,Z 614.146,A -85,B 0,C 180,E1 -24946.514,E2 -24946.514} C_VEL
LIN {X 0,Y 129.59,Z 611.184,A -85,B 0,C 180,E1 -24948.802,E2 -24948.802} C_VEL
LIN {X 0,Y 132.311,Z 603.653,A -85,B 0,C 180,E1 -24953.477,E2 -24953.477} C_VEL
LIN {X 0,Y 135.033,Z 596.222,A -85,B 0,C 180,E1 -24957.091,E2 -24957.091} C_VEL
LIN {X 0,Y 137.367,Z 589.169,A -85,B 0,C 180,E1 -24959.915,E2 -24959.915} C_VEL
LIN {X 0,Y 140.869,Z 578.41,A -85,B 0,C 180,E1 -24963.284,E2 -24963.284} C_VEL
LIN {X 0,Y 143.669,Z 569.187,A -85,B 0,C 180,E1 -24965.514,E2 -24965.514} C_VEL
LIN {X 0,Y 146.696,Z 557.771,A -85,B 0,C 180,E1 -24967.65,E2 -24967.65} C_VEL
LIN {X 0,Y 149.138,Z 546.038,A -85,B 0,C 180,E1 -24969.289,E2 -24969.289} C_VEL
LIN {X 0,Y 151.135,Z 533.426,A -85,B 0,C 180,E1 -24970.509,E2 -24970.509} C_VEL
LIN {X 0,Y 152.495,Z 519.806,A -85,B 0,C 180,E1 -24971.33,E2 -24971.33} C_VEL
LIN {X 0,Y 155.101,Z 475.55,A -85,B 0,C 180,E1 -24973.166,E2 -24973.166} C_VEL
LIN {X 0,Y 154.633,Z 472.352,A -85,B 0,C 180,E1 -24973.484,E2 -24973.484} C_VEL
LIN {X 0,Y 149.493,Z 457.719,A -85,B 0,C 180,E1 -24975.929,E2 -24975.929} C_VEL
LIN {X 0,Y 145.243,Z 448.19,A -85,B 0,C 180,E1 -24977.978,E2 -24977.978} C_VEL
LIN {X 0,Y 139.905,Z 439.266,A -85,B 0,C 180,E1 -24980.62,E2 -24980.62} C_VEL
LIN {X 0,Y 134.912,Z 432.065,A -85,B 0,C 180,E1 -24983.312,E2 -24983.312} C_VEL
LIN {X 0,Y 132.688,Z 428.845,A -85,B 0,C 180,E1 -24984.623,E2 -24984.623} C_VEL
LIN {X 0,Y 131.858,Z 427.738,A -85,B 0,C 180,E1 -24985.126,E2 -24985.126} C_VEL
LIN {X 0,Y 129.808,Z 425.388,A -85,B 0,C 180,E1 -24986.383,E2 -24986.383} C_VEL
LIN {X 0,Y 129.077,Z 423.389,A -85,B 0,C 180,E1 -24987.243,E2 -24987.243} C_VEL
LIN {X 0,Y 129.006,Z 422.969,A -85,B 0,C 180,E1 -24987.916,E2 -24987.916} C_VEL
LIN {X 0,Y 129.027,Z 422.903,A -85,B 0,C 180,E1 -24994.166,E2 -24994.166} C_VEL
LIN {X 0,Y 129.107,Z 422.873,A -85,B 0,C 180,E1 -24997.728,E2 -24997.728} C_VEL
LIN {X 0,Y 129.183,Z 422.894,A -85,B 0,C 180,E1 -25004.215,E2 -25004.215} C_VEL
LIN {X 0,Y 129.389,Z 422.827,A -85,B 0,C 180,E1 -25007.877,E2 -25007.877} C_VEL
LIN {X 0,Y 129.466,Z 422.811,A -85,B 0,C 180,E1 -25010.627,E2 -25010.627} C_VEL
LIN {X 0,Y 129.671,Z 422.817,A -85,B 0,C 180,E1 -25016.893,E2 -25016.893} C_VEL
LIN {X 0,Y 130.087,Z 422.728,A -85,B 0,C 180,E1 -25020,E2 -25020} C_VEL
LIN {X 0,Y 129.446,Z 422.848,A -85,B 0,C 180,E1 -25027.021,E2 -25027.021} C_VEL
LIN {X 0,Y 129.347,Z 422.818,A -85,B 0,C 180,E1 -25032.038,E2 -25032.038} C_VEL
LIN {X 0,Y 129.151,Z 422.893,A -85,B 0,C 180,E1 -25039.056,E2 -25039.056} C_VEL
LIN {X 0,Y 129.108,Z 422.856,A -85,B 0,C 180,E1 -25042.398,E2 -25042.398} C_VEL
LIN {X 0,Y 129.036,Z 422.908,A -85,B 0,C 180,E1 -25049.373,E2 -25049.373} C_VEL
LIN {X 0,Y 128.96,Z 422.885,A -85,B 0,C 180,E1 -25055.169,E2 -25055.169} C_VEL
LIN {X 0,Y 128.935,Z 422.896,A -85,B 0,C 180,E1 -25060.851,E2 -25060.851} C_VEL
LIN {X 0,Y 128.99,Z 423.152,A -85,B 0,C 180,E1 -25065.722,E2 -25065.722} C_VEL
LIN {X 0,Y 129.316,Z 424.341,A -85,B 0,C 180,E1 -25066.485,E2 -25066.485} C_VEL
LIN {X 0,Y 130.727,Z 426.734,A -85,B 0,C 180,E1 -25067.47,E2 -25067.47} C_VEL
LIN {X 0,Y 132.526,Z 428.539,A -85,B 0,C 180,E1 -25068.528,E2 -25068.528} C_VEL
LIN {X 0,Y 134.749,Z 431.895,A -85,B 0,C 180,E1 -25069.855,E2 -25069.855} C_VEL
LIN {X 0,Y 136.114,Z 433.696,A -85,B 0,C 180,E1 -25070.613,E2 -25070.613} C_VEL
LIN {X 0,Y 140.854,Z 440.779,A -85,B 0,C 180,E1 -25073.124,E2 -25073.124} C_VEL
LIN {X 0,Y 146.55,Z 450.415,A -85,B 0,C 180,E1 -25075.882,E2 -25075.882} C_VEL
LIN {X 0,Y 151.609,Z 460.235,A -85,B 0,C 180,E1 -25078.149,E2 -25078.149} C_VEL
LIN {X 0,Y 155.398,Z 471.29,A -85,B 0,C 180,E1 -25079.928,E2 -25079.928} C_VEL
LIN {X 0,Y 152.081,Z 522.153,A -85,B 0,C 180,E1 -25082.032,E2 -25082.032} C_VEL
LIN {X 0,Y 150.376,Z 535.779,A -85,B 0,C 180,E1 -25083.075,E2 -25083.075} C_VEL
LIN {X 0,Y 148.22,Z 547.739,A -85,B 0,C 180,E1 -25084.453,E2 -25084.453} C_VEL
LIN {X 0,Y 145.478,Z 559.915,A -85,B 0,C 180,E1 -25086.436,E2 -25086.436} C_VEL
LIN {X 0,Y 142.542,Z 570.392,A -85,B 0,C 180,E1 -25088.677,E2 -25088.677} C_VEL
LIN {X 0,Y 139.454,Z 579.883,A -85,B 0,C 180,E1 -25091.259,E2 -25091.259} C_VEL
LIN {X 0,Y 136.514,Z 588.665,A -85,B 0,C 180,E1 -25094.319,E2 -25094.319} C_VEL
LIN {X 0,Y 133.677,Z 596.742,A -85,B 0,C 180,E1 -25097.86,E2 -25097.86} C_VEL
LIN {X 0,Y 130.773,Z 604.682,A -85,B 0,C 180,E1 -25102.278,E2 -25102.278} C_VEL
LIN {X 0,Y 128.703,Z 611.001,A -85,B 0,C 180,E1 -25106.869,E2 -25106.869} C_VEL
LIN {X 0,Y 127.317,Z 616.032,A -85,B 0,C 180,E1 -25111.581,E2 -25111.581} C_VEL
LIN {X 0,Y 126.382,Z 619.94,A -85,B 0,C 180,E1 -25116.385,E2 -25116.385} C_VEL
LIN {X 0,Y 125.976,Z 621.961,A -85,B 0,C 180,E1 -25119.634,E2 -25119.634} C_VEL
LIN {X 0,Y 125.851,Z 623.561,A -85,B 0,C 180,E1 -25122.906,E2 -25122.906} C_VEL
LIN {X 0,Y 126.357,Z 625.35,A -85,B 0,C 180,E1 -25128.996,E2 -25128.996} C_VEL
LIN {X 0,Y 127.043,Z 625.747,A -85,B 0,C 180,E1 -25132.781,E2 -25132.781} C_VEL
LIN {X 0,Y 128.047,Z 625.66,A -85,B 0,C 180,E1 -25136.044,E2 -25136.044} C_VEL
LIN {X 0,Y 129.729,Z 624.943,A -85,B 0,C 180,E1 -25139.913,E2 -25139.913} C_VEL
LIN {X 0,Y 133.142,Z 622.769,A -85,B 0,C 180,E1 -25145.494,E2 -25145.494} C_VEL
LIN {X 0,Y 136.479,Z 620.18,A -85,B 0,C 180,E1 -25149.428,E2 -25149.428} C_VEL
LIN {X 0,Y 141.399,Z 615.759,A -85,B 0,C 180,E1 -25154.093,E2 -25154.093} C_VEL
LIN {X 0,Y 147.048,Z 609.949,A -85,B 0,C 180,E1 -25158.305,E2 -25158.305} C_VEL
LIN {X 0,Y 153.474,Z 602.461,A -85,B 0,C 180,E1 -25162.176,E2 -25162.176} C_VEL
LIN {X 0,Y 159.516,Z 594.459,A -85,B 0,C 180,E1 -25165.201,E2 -25165.201} C_VEL
LIN {X 0,Y 165.79,Z 584.642,A -85,B 0,C 180,E1 -25167.972,E2 -25167.972} C_VEL
LIN {X 0,Y 171.415,Z 574.394,A -85,B 0,C 180,E1 -25170.123,E2 -25170.123} C_VEL
LIN {X 0,Y 176.292,Z 563.53,A -85,B 0,C 180,E1 -25171.885,E2 -25171.885} C_VEL
LIN {X 0,Y 180.487,Z 551.986,A -85,B 0,C 180,E1 -25173.27,E2 -25173.27} C_VEL
LIN {X 0,Y 184.125,Z 539.257,A -85,B 0,C 180,E1 -25174.343,E2 -25174.343} C_VEL
LIN {X 0,Y 186.715,Z 526.162,A -85,B 0,C 180,E1 -25175.092,E2 -25175.092} C_VEL
LIN {X 0,Y 188.434,Z 510.266,A -85,B 0,C 180,E1 -25175.649,E2 -25175.649} C_VEL
LIN {X 0,Y 189.206,Z 500.714,A -85,B 0,C 180,E1 -25175.957,E2 -25175.957} C_VEL
LIN {X 0,Y 185.568,Z 492.219,A -85,B 0,C 180,E1 -25178.549,E2 -25178.549} C_VEL
LIN {X 0,Y 181.517,Z 483.809,A -85,B 0,C 180,E1 -25181.774,E2 -25181.774} C_VEL
LIN {X 0,Y 177.792,Z 477.716,A -85,B 0,C 180,E1 -25185.115,E2 -25185.115} C_VEL
LIN {X 0,Y 174.893,Z 473.285,A -85,B 0,C 180,E1 -25188.181,E2 -25188.181} C_VEL
LIN {X 0,Y 172.458,Z 469.425,A -85,B 0,C 180,E1 -25191.357,E2 -25191.357} C_VEL
LIN {X 0,Y 170.159,Z 465.786,A -85,B 0,C 180,E1 -25195.262,E2 -25195.262} C_VEL
LIN {X 0,Y 169.822,Z 465.106,A -85,B 0,C 180,E1 -25195.996,E2 -25195.996} C_VEL
LIN {X 0,Y 167.686,Z 462.549,A -85,B 0,C 180,E1 -25202.402,E2 -25202.402} C_VEL
LIN {X 0,Y 167.345,Z 462.304,A -85,B 0,C 180,E1 -25207.969,E2 -25207.969} C_VEL
LIN {X 0,Y 169.772,Z 465.444,A -85,B 0,C 180,E1 -25216.845,E2 -25216.845} C_VEL
LIN {X 0,Y 171.796,Z 469.02,A -85,B 0,C 180,E1 -25220.599,E2 -25220.599} C_VEL
LIN {X 0,Y 172.966,Z 470.34,A -85,B 0,C 180,E1 -25222.239,E2 -25222.239} C_VEL
LIN {X 0,Y 175.745,Z 474.968,A -85,B 0,C 180,E1 -25225.677,E2 -25225.677} C_VEL
LIN {X 0,Y 178.677,Z 480.457,A -85,B 0,C 180,E1 -25228.721,E2 -25228.721} C_VEL
LIN {X 0,Y 181.647,Z 486.212,A -85,B 0,C 180,E1 -25231.387,E2 -25231.387} C_VEL
LIN {X 0,Y 186.266,Z 496.641,A -85,B 0,C 180,E1 -25235.045,E2 -25235.045} C_VEL
LIN {X 0,Y 188.984,Z 503.558,A -85,B 0,C 180,E1 -25236.991,E2 -25236.991} C_VEL
LIN {X 0,Y 186.95,Z 526.048,A -85,B 0,C 180,E1 -25237.749,E2 -25237.749} C_VEL
LIN {X 0,Y 184.541,Z 539.472,A -85,B 0,C 180,E1 -25238.443,E2 -25238.443} C_VEL
LIN {X 0,Y 181.646,Z 550.654,A -85,B 0,C 180,E1 -25239.305,E2 -25239.305} C_VEL
LIN {X 0,Y 177.721,Z 561.934,A -85,B 0,C 180,E1 -25240.428,E2 -25240.428} C_VEL
LIN {X 0,Y 172.733,Z 573.541,A -85,B 0,C 180,E1 -25242.054,E2 -25242.054} C_VEL
LIN {X 0,Y 167.333,Z 583.979,A -85,B 0,C 180,E1 -25244.01,E2 -25244.01} C_VEL
LIN {X 0,Y 162.28,Z 592.512,A -85,B 0,C 180,E1 -25246.14,E2 -25246.14} C_VEL
LIN {X 0,Y 156.805,Z 600.409,A -85,B 0,C 180,E1 -25248.618,E2 -25248.618} C_VEL
LIN {X 0,Y 150.683,Z 608.168,A -85,B 0,C 180,E1 -25251.832,E2 -25251.832} C_VEL
LIN {X 0,Y 145.276,Z 614.346,A -85,B 0,C 180,E1 -25255.327,E2 -25255.327} C_VEL
LIN {X 0,Y 139.615,Z 620.057,A -85,B 0,C 180,E1 -25259.777,E2 -25259.777} C_VEL
LIN {X 0,Y 135.5,Z 623.743,A -85,B 0,C 180,E1 -25263.842,E2 -25263.842} C_VEL
LIN {X 0,Y 132.032,Z 626.441,A -85,B 0,C 180,E1 -25268.125,E2 -25268.125} C_VEL
LIN {X 0,Y 128.807,Z 628.625,A -85,B 0,C 180,E1 -25274.17,E2 -25274.17} C_VEL
LIN {X 0,Y 127.712,Z 629.119,A -85,B 0,C 180,E1 -25277.285,E2 -25277.285} C_VEL
LIN {X 0,Y 126.522,Z 628.921,A -85,B 0,C 180,E1 -25283.622,E2 -25283.622} C_VEL
LIN {X 0,Y 126.311,Z 628.253,A -85,B 0,C 180,E1 -25286.811,E2 -25286.811} C_VEL
LIN {X 0,Y 126.39,Z 627.188,A -85,B 0,C 180,E1 -25290.001,E2 -25290.001} C_VEL
LIN {X 0,Y 126.304,Z 625.658,A -85,B 0,C 180,E1 -25293.191,E2 -25293.191} C_VEL
LIN {X 0,Y 126.58,Z 622.564,A -85,B 0,C 180,E1 -25297.979,E2 -25297.979} C_VEL
LIN {X 0,Y 127.464,Z 618.389,A -85,B 0,C 180,E1 -25302.742,E2 -25302.742} C_VEL
LIN {X 0,Y 129.319,Z 611.99,A -85,B 0,C 180,E1 -25308.21,E2 -25308.21} C_VEL
LIN {X 0,Y 129.59,Z 611.184,A -85,B 0,C 180,E1 -25308.802,E2 -25308.802} C_VEL
LIN {X 0,Y 130.02,Z 608.066,A -85,B 0,C 180,E1 -25311.019,E2 -25311.019} C_VEL
LIN {X 0,Y 129.226,Z 602.51,A -85,B 0,C 180,E1 -25314.654,E2 -25314.654} C_VEL
LIN {X 0,Y 128.792,Z 596.325,A -85,B 0,C 180,E1 -25318.113,E2 -25318.113} C_VEL
LIN {X 0,Y 129.744,Z 592.221,A -85,B 0,C 180,E1 -25319.96,E2 -25319.96} C_VEL
LIN {X 0,Y 133.371,Z 582.028,A -85,B 0,C 180,E1 -25323.594,E2 -25323.594} C_VEL
LIN {X 0,Y 136.999,Z 570.814,A -85,B 0,C 180,E1 -25326.61,E2 -25326.61} C_VEL
LIN {X 0,Y 140.219,Z 559.834,A -85,B 0,C 180,E1 -25328.794,E2 -25328.794} C_VEL
LIN {X 0,Y 142.967,Z 547.628,A -85,B 0,C 180,E1 -25330.643,E2 -25330.643} C_VEL
LIN {X 0,Y 145.127,Z 534.991,A -85,B 0,C 180,E1 -25331.982,E2 -25331.982} C_VEL
LIN {X 0,Y 146.659,Z 521.476,A -85,B 0,C 180,E1 -25332.857,E2 -25332.857} C_VEL
LIN {X 0,Y 149.444,Z 476.006,A -85,B 0,C 180,E1 -25334.816,E2 -25334.816} C_VEL
LIN {X 0,Y 145.716,Z 464.364,A -85,B 0,C 180,E1 -25336.757,E2 -25336.757} C_VEL
LIN {X 0,Y 141.5,Z 454.057,A -85,B 0,C 180,E1 -25338.956,E2 -25338.956} C_VEL
LIN {X 0,Y 136.617,Z 445.252,A -85,B 0,C 180,E1 -25341.553,E2 -25341.553} C_VEL
LIN {X 0,Y 131.098,Z 437.214,A -85,B 0,C 180,E1 -25344.723,E2 -25344.723} C_VEL
LIN {X 0,Y 128.356,Z 433.278,A -85,B 0,C 180,E1 -25346.474,E2 -25346.474} C_VEL
LIN {X 0,Y 126.078,Z 430.191,A -85,B 0,C 180,E1 -25348.024,E2 -25348.024} C_VEL
LIN {X 0,Y 125.389,Z 429.024,A -85,B 0,C 180,E1 -25348.536,E2 -25348.536} C_VEL
LIN {X 0,Y 123.017,Z 426.692,A -85,B 0,C 180,E1 -25350.226,E2 -25350.226} C_VEL
LIN {X 0,Y 122.044,Z 424.404,A -85,B 0,C 180,E1 -25351.357,E2 -25351.357} C_VEL
LIN {X 0,Y 121.94,Z 423.822,A -85,B 0,C 180,E1 -25352.543,E2 -25352.543} C_VEL
LIN {X 0,Y 122.028,Z 423.759,A -85,B 0,C 180,E1 -25357.145,E2 -25357.145} C_VEL
LIN {X 0,Y 122.095,Z 423.763,A -85,B 0,C 180,E1 -25363.273,E2 -25363.273} C_VEL
LIN {X 0,Y 122.312,Z 423.709,A -85,B 0,C 180,E1 -25367.637,E2 -25367.637} C_VEL
LIN {X 0,Y 122.42,Z 423.717,A -85,B 0,C 180,E1 -25373.407,E2 -25373.407} C_VEL
LIN {X 0,Y 123.041,Z 423.604,A -85,B 0,C 180,E1 -25380,E2 -25380} C_VEL
LIN {X 0,Y 122.403,Z 423.731,A -85,B 0,C 180,E1 -25386.938,E2 -25386.938} C_VEL
LIN {X 0,Y 122.289,Z 423.695,A -85,B 0,C 180,E1 -25392.315,E2 -25392.315} C_VEL
LIN {X 0,Y 122.099,Z 423.76,A -85,B 0,C 180,E1 -25396.726,E2 -25396.726} C_VEL
LIN {X 0,Y 122.022,Z 423.735,A -85,B 0,C 180,E1 -25402.849,E2 -25402.849} C_VEL
LIN {X 0,Y 121.957,Z 423.774,A -85,B 0,C 180,E1 -25407.452,E2 -25407.452} C_VEL
LIN {X 0,Y 121.904,Z 423.769,A -85,B 0,C 180,E1 -25411.256,E2 -25411.256} C_VEL
LIN {X 0,Y 121.885,Z 423.775,A -85,B 0,C 180,E1 -25416.172,E2 -25416.172} C_VEL
LIN {X 0,Y 121.89,Z 423.86,A -85,B 0,C 180,E1 -25421.152,E2 -25421.152} C_VEL
LIN {X 0,Y 122.033,Z 424.788,A -85,B 0,C 180,E1 -25422.113,E2 -25422.113} C_VEL
LIN {X 0,Y 123.41,Z 427.45,A -85,B 0,C 180,E1 -25423.356,E2 -25423.356} C_VEL
LIN {X 0,Y 125.741,Z 429.559,A -85,B 0,C 180,E1 -25424.978,E2 -25424.978} C_VEL
LIN {X 0,Y 127.822,Z 432.79,A -85,B 0,C 180,E1 -25426.45,E2 -25426.45} C_VEL
